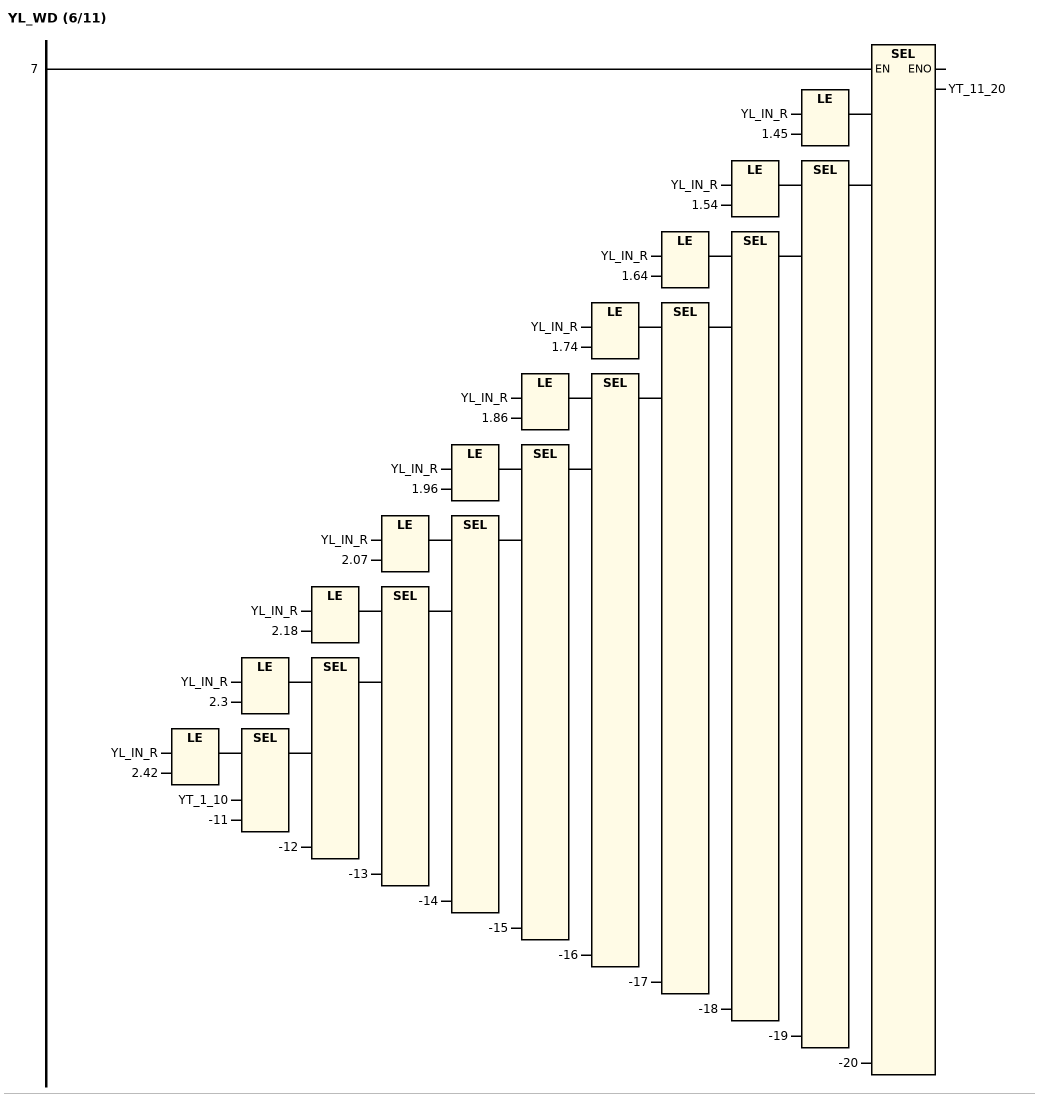
[picture p48: YL_WD (LD)]
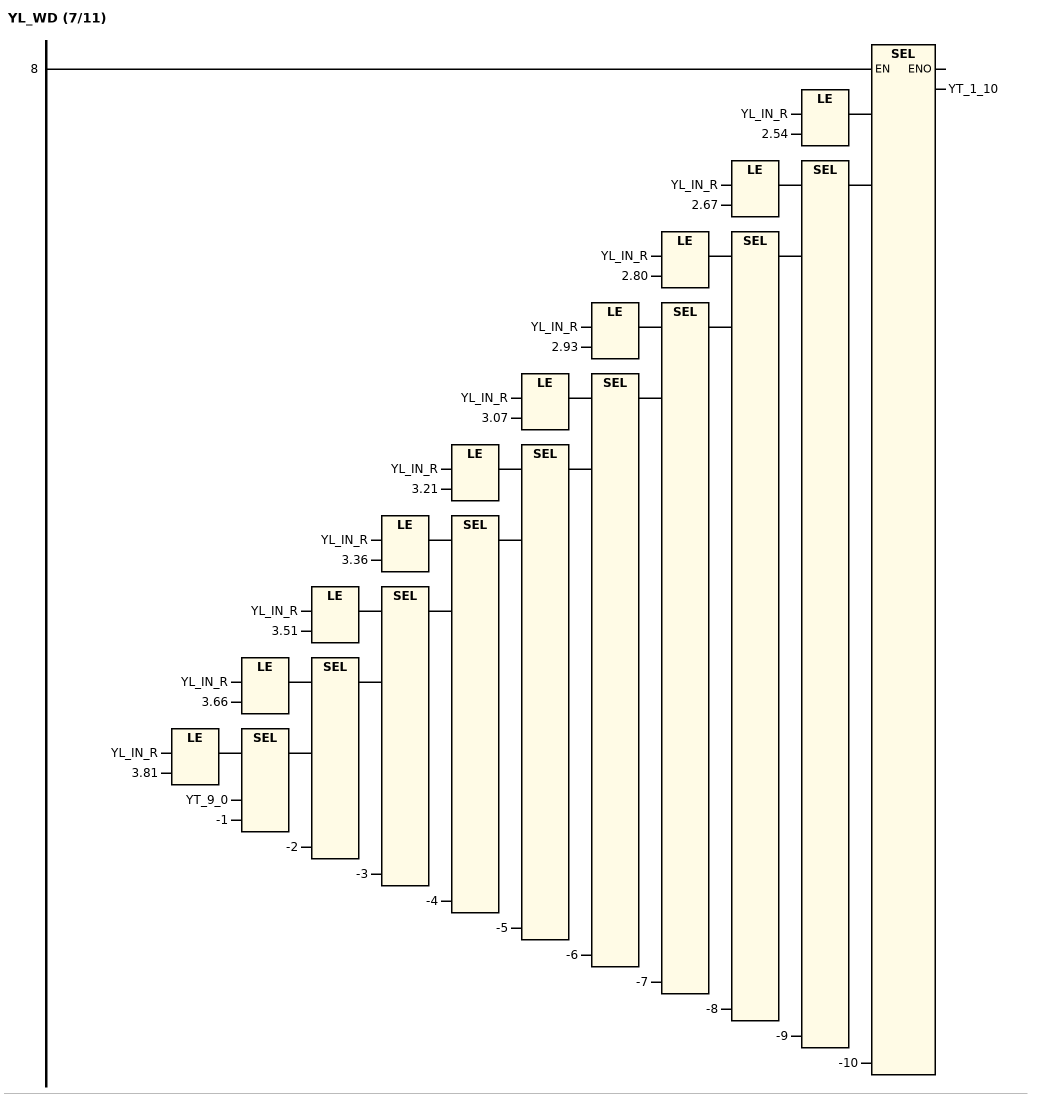
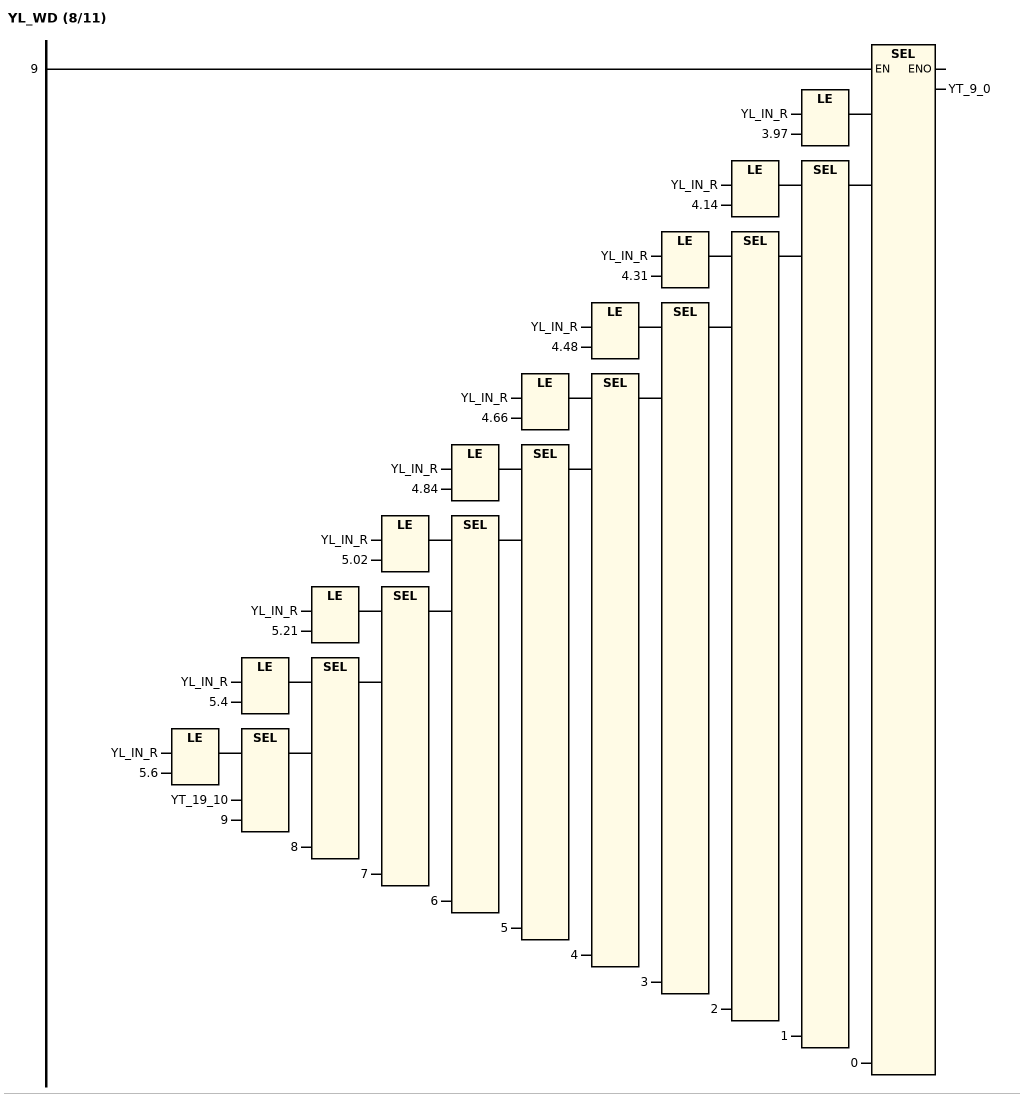
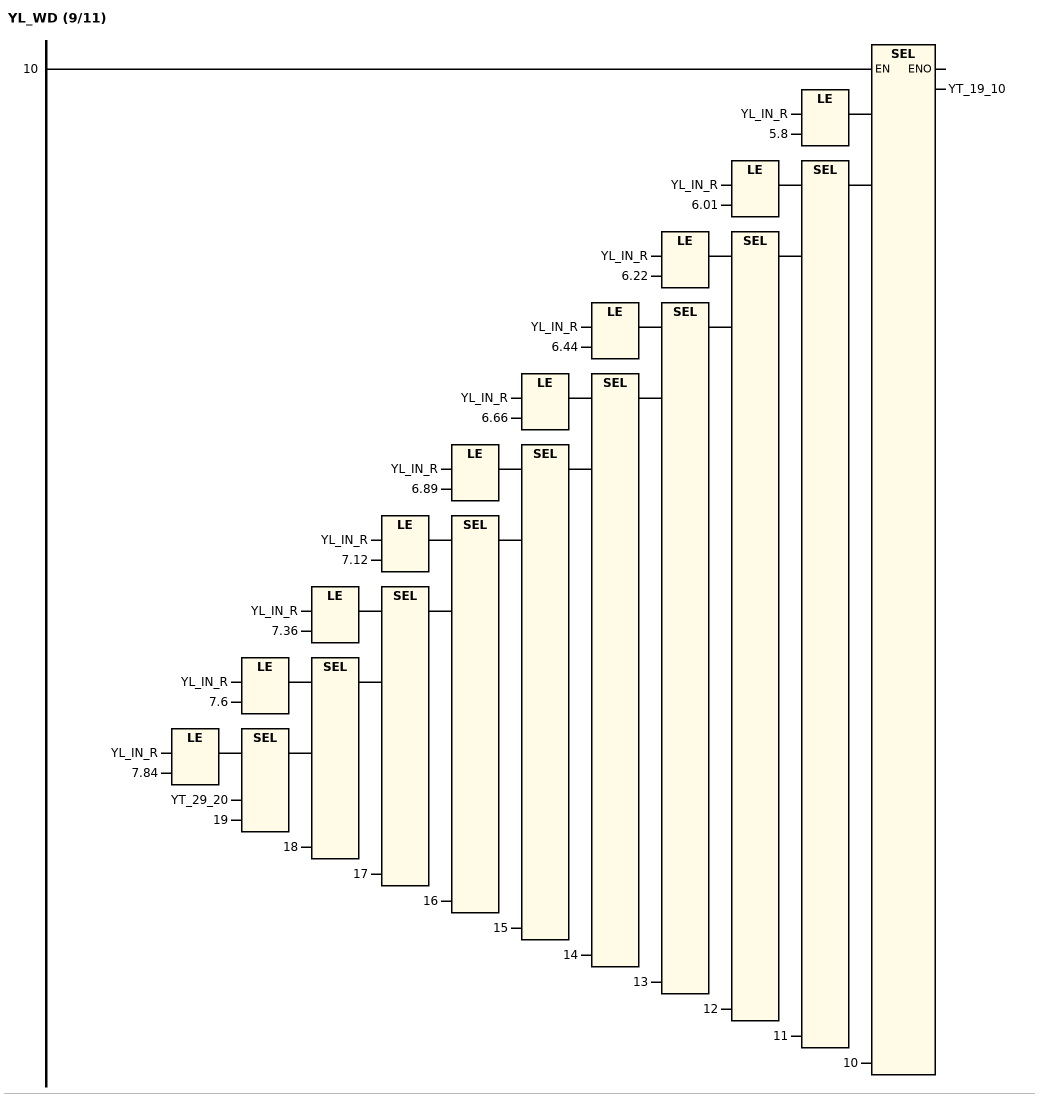
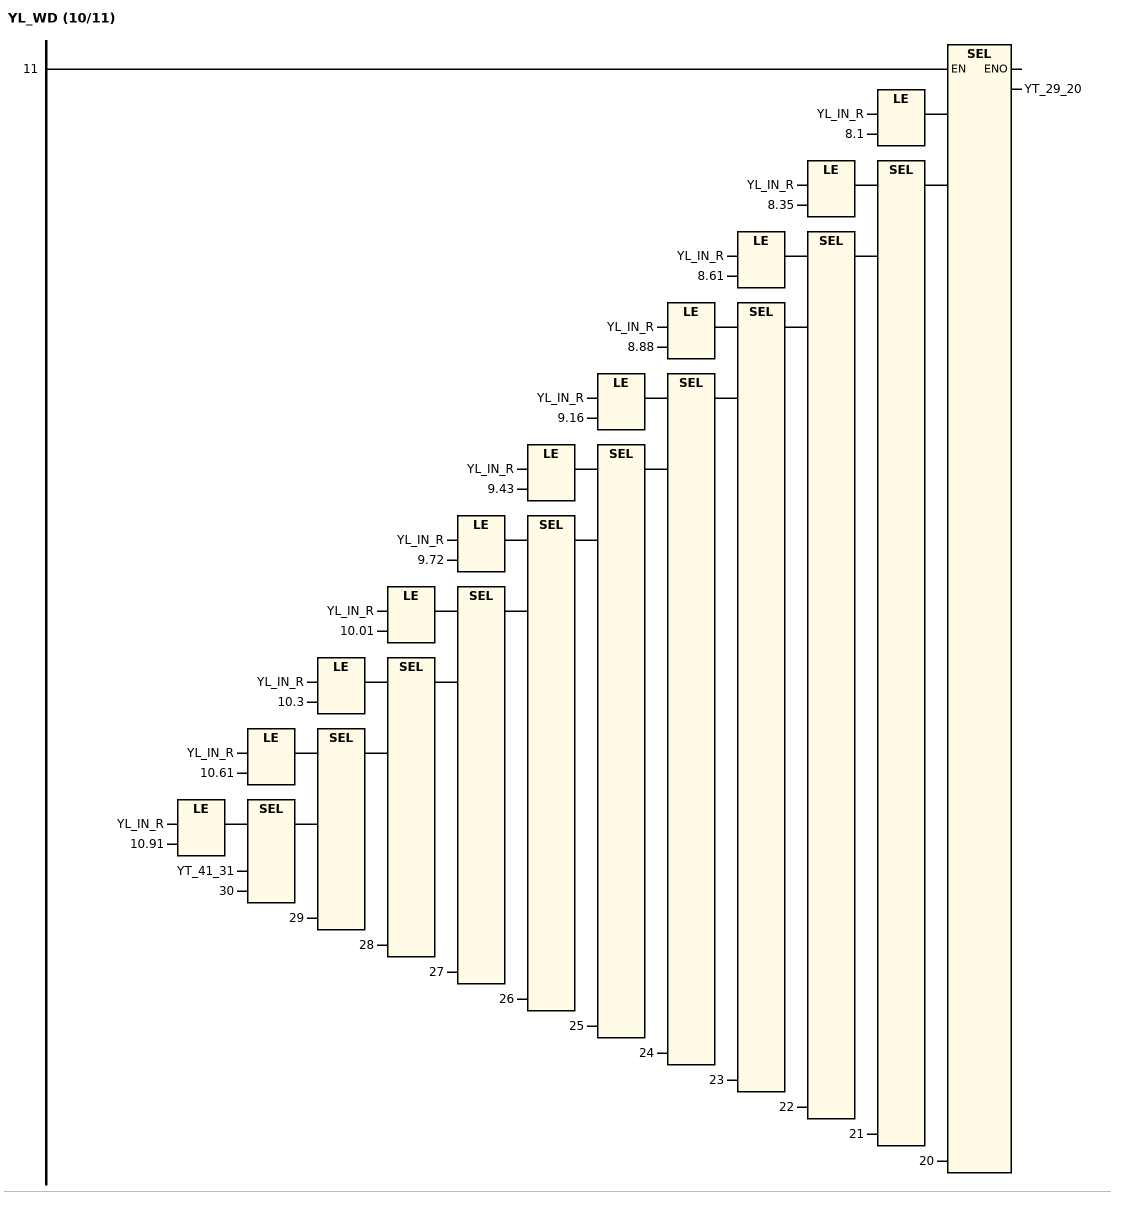
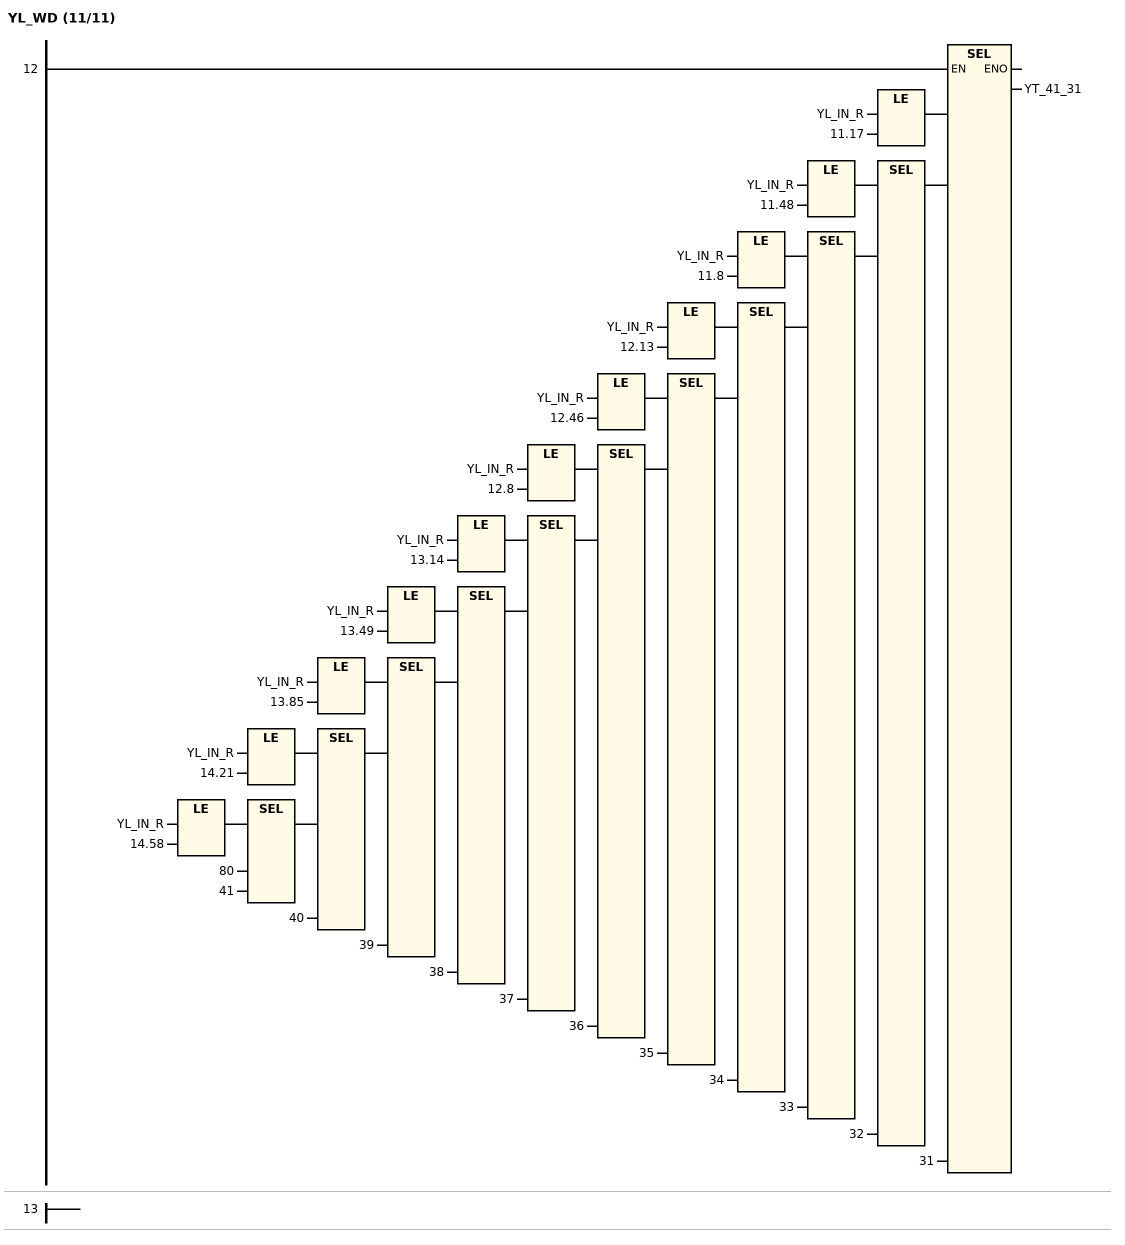
_LD_ (* Ladder Diagram *)
NETWORK 1
	*
		EN --- DIV(INT_TO_REAL(YL_IN), 100) => YL_IN_R
NETWORK 2
	*
		EN --- MUL(YL_T_KA, 10) => YL_T
NETWORK 3
	*
		EN --- SEL(LE(YL_IN_R, -0.62), SEL(LE(YL_IN_R, -0.60), SEL(LE(YL_IN_R, -0.58), SEL(LE(YL_IN_R, -0.55), SEL(LE(YL_IN_R, -0.53), SEL(LE(YL_IN_R, -0.50), SEL(LE(YL_IN_R, -0.46), SEL(LE(YL_IN_R, -0.44), SEL(LE(YL_IN_R, -0.41), SEL(LE(YL_IN_R, -0.38), YT_51_60, -51), -52), -53), -54), -55), -56), -57), -58), -59), -60) => YL_T_KA
NETWORK 4
	*
		EN --- SEL(LE(YL_IN_R, -0.35), SEL(LE(YL_IN_R, -0.32), SEL(LE(YL_IN_R, -0.28), SEL(LE(YL_IN_R, -0.24), SEL(LE(YL_IN_R, -0.21), SEL(LE(YL_IN_R, -0.17), SEL(LE(YL_IN_R, -0.12), SEL(LE(YL_IN_R, -0.08), SEL(LE(YL_IN_R, -0.04), SEL(LE(YL_IN_R, 0.00), YT_41_50, -41), -42), -43), -44), -45), -46), -47), -48), -49), -50) => YT_51_60
NETWORK 5
	*
		EN --- SEL(LE(YL_IN_R, 0.05), SEL(LE(YL_IN_R, 0.1), SEL(LE(YL_IN_R, 0.15), SEL(LE(YL_IN_R, 0.2), SEL(LE(YL_IN_R, 0.26), SEL(LE(YL_IN_R, 0.32), SEL(LE(YL_IN_R, 0.37), SEL(LE(YL_IN_R, 0.44), SEL(LE(YL_IN_R, 0.5), SEL(LE(YL_IN_R, 0.57), YT_31_40, -31), -32), -33), -34), -35), -36), -37), -38), -39), -40) => YT_41_50
NETWORK 6
	*
		EN --- SEL(LE(YL_IN_R, 0.63), SEL(LE(YL_IN_R, 0.70), SEL(LE(YL_IN_R, 0.78), SEL(LE(YL_IN_R, 0.85), SEL(LE(YL_IN_R, 0.93), SEL(LE(YL_IN_R, 1.01), SEL(LE(YL_IN_R, 1.09), SEL(LE(YL_IN_R, 1.18), SEL(LE(YL_IN_R, 1.26), SEL(LE(YL_IN_R, 1.36), YT_11_20, -21), -22), -23), -24), -25), -26), -27), -28), -29), -30) => YT_31_40
NETWORK 7
	*
		EN --- SEL(LE(YL_IN_R, 1.45), SEL(LE(YL_IN_R, 1.54), SEL(LE(YL_IN_R, 1.64), SEL(LE(YL_IN_R, 1.74), SEL(LE(YL_IN_R, 1.86), SEL(LE(YL_IN_R, 1.96), SEL(LE(YL_IN_R, 2.07), SEL(LE(YL_IN_R, 2.18), SEL(LE(YL_IN_R, 2.3), SEL(LE(YL_IN_R, 2.42), YT_1_10, -11), -12), -13), -14), -15), -16), -17), -18), -19), -20) => YT_11_20
NETWORK 8
	*
		EN --- SEL(LE(YL_IN_R, 2.54), SEL(LE(YL_IN_R, 2.67), SEL(LE(YL_IN_R, 2.80), SEL(LE(YL_IN_R, 2.93), SEL(LE(YL_IN_R, 3.07), SEL(LE(YL_IN_R, 3.21), SEL(LE(YL_IN_R, 3.36), SEL(LE(YL_IN_R, 3.51), SEL(LE(YL_IN_R, 3.66), SEL(LE(YL_IN_R, 3.81), YT_9_0, -1), -2), -3), -4), -5), -6), -7), -8), -9), -10) => YT_1_10
NETWORK 9
	*
		EN --- SEL(LE(YL_IN_R, 3.97), SEL(LE(YL_IN_R, 4.14), SEL(LE(YL_IN_R, 4.31), SEL(LE(YL_IN_R, 4.48), SEL(LE(YL_IN_R, 4.66), SEL(LE(YL_IN_R, 4.84), SEL(LE(YL_IN_R, 5.02), SEL(LE(YL_IN_R, 5.21), SEL(LE(YL_IN_R, 5.4), SEL(LE(YL_IN_R, 5.6), YT_19_10, 9), 8), 7), 6), 5), 4), 3), 2), 1), 0) => YT_9_0
NETWORK 10
	*
		EN --- SEL(LE(YL_IN_R, 5.8), SEL(LE(YL_IN_R, 6.01), SEL(LE(YL_IN_R, 6.22), SEL(LE(YL_IN_R, 6.44), SEL(LE(YL_IN_R, 6.66), SEL(LE(YL_IN_R, 6.89), SEL(LE(YL_IN_R, 7.12), SEL(LE(YL_IN_R, 7.36), SEL(LE(YL_IN_R, 7.6), SEL(LE(YL_IN_R, 7.84), YT_29_20, 19), 18), 17), 16), 15), 14), 13), 12), 11), 10) => YT_19_10
NETWORK 11
	*
		EN --- SEL(LE(YL_IN_R, 8.1), SEL(LE(YL_IN_R, 8.35), SEL(LE(YL_IN_R, 8.61), SEL(LE(YL_IN_R, 8.88), SEL(LE(YL_IN_R, 9.16), SEL(LE(YL_IN_R, 9.43), SEL(LE(YL_IN_R, 9.72), SEL(LE(YL_IN_R, 10.01), SEL(LE(YL_IN_R, 10.3), SEL(LE(YL_IN_R, 10.61), SEL(LE(YL_IN_R, 10.91), YT_41_31, 30), 29), 28), 27), 26), 25), 24), 23), 22), 21), 20) => YT_29_20
NETWORK 12
	*
		EN --- SEL(LE(YL_IN_R, 11.17), SEL(LE(YL_IN_R, 11.48), SEL(LE(YL_IN_R, 11.8), SEL(LE(YL_IN_R, 12.13), SEL(LE(YL_IN_R, 12.46), SEL(LE(YL_IN_R, 12.8), SEL(LE(YL_IN_R, 13.14), SEL(LE(YL_IN_R, 13.49), SEL(LE(YL_IN_R, 13.85), SEL(LE(YL_IN_R, 14.21), SEL(LE(YL_IN_R, 14.58), 80, 41), 40), 39), 38), 37), 36), 35), 34), 33), 32), 31) => YT_41_31
NETWORK 13
	*
_END_LD_
(* the same logic as Structured Text *)
(* Network 1 *)
YL_IN_R := INT_TO_REAL(YL_IN) / 100;
(* Network 2 *)
YL_T := YL_T_KA * 10;
(* Network 3 *)
YL_T_KA := SEL(YL_IN_R <= (-0.62), SEL(YL_IN_R <= (-0.60), SEL(YL_IN_R <= (-0.58), SEL(YL_IN_R <= (-0.55), SEL(YL_IN_R <= (-0.53), SEL(YL_IN_R <= (-0.50), SEL(YL_IN_R <= (-0.46), SEL(YL_IN_R <= (-0.44), SEL(YL_IN_R <= (-0.41), SEL(YL_IN_R <= (-0.38), YT_51_60, -51), -52), -53), -54), -55), -56), -57), -58), -59), -60);
(* Network 4 *)
YT_51_60 := SEL(YL_IN_R <= (-0.35), SEL(YL_IN_R <= (-0.32), SEL(YL_IN_R <= (-0.28), SEL(YL_IN_R <= (-0.24), SEL(YL_IN_R <= (-0.21), SEL(YL_IN_R <= (-0.17), SEL(YL_IN_R <= (-0.12), SEL(YL_IN_R <= (-0.08), SEL(YL_IN_R <= (-0.04), SEL(YL_IN_R <= 0.00, YT_41_50, -41), -42), -43), -44), -45), -46), -47), -48), -49), -50);
(* Network 5 *)
YT_41_50 := SEL(YL_IN_R <= 0.05, SEL(YL_IN_R <= 0.1, SEL(YL_IN_R <= 0.15, SEL(YL_IN_R <= 0.2, SEL(YL_IN_R <= 0.26, SEL(YL_IN_R <= 0.32, SEL(YL_IN_R <= 0.37, SEL(YL_IN_R <= 0.44, SEL(YL_IN_R <= 0.5, SEL(YL_IN_R <= 0.57, YT_31_40, -31), -32), -33), -34), -35), -36), -37), -38), -39), -40);
(* Network 6 *)
YT_31_40 := SEL(YL_IN_R <= 0.63, SEL(YL_IN_R <= 0.70, SEL(YL_IN_R <= 0.78, SEL(YL_IN_R <= 0.85, SEL(YL_IN_R <= 0.93, SEL(YL_IN_R <= 1.01, SEL(YL_IN_R <= 1.09, SEL(YL_IN_R <= 1.18, SEL(YL_IN_R <= 1.26, SEL(YL_IN_R <= 1.36, YT_11_20, -21), -22), -23), -24), -25), -26), -27), -28), -29), -30);
(* Network 7 *)
YT_11_20 := SEL(YL_IN_R <= 1.45, SEL(YL_IN_R <= 1.54, SEL(YL_IN_R <= 1.64, SEL(YL_IN_R <= 1.74, SEL(YL_IN_R <= 1.86, SEL(YL_IN_R <= 1.96, SEL(YL_IN_R <= 2.07, SEL(YL_IN_R <= 2.18, SEL(YL_IN_R <= 2.3, SEL(YL_IN_R <= 2.42, YT_1_10, -11), -12), -13), -14), -15), -16), -17), -18), -19), -20);
(* Network 8 *)
YT_1_10 := SEL(YL_IN_R <= 2.54, SEL(YL_IN_R <= 2.67, SEL(YL_IN_R <= 2.80, SEL(YL_IN_R <= 2.93, SEL(YL_IN_R <= 3.07, SEL(YL_IN_R <= 3.21, SEL(YL_IN_R <= 3.36, SEL(YL_IN_R <= 3.51, SEL(YL_IN_R <= 3.66, SEL(YL_IN_R <= 3.81, YT_9_0, -1), -2), -3), -4), -5), -6), -7), -8), -9), -10);
(* Network 9 *)
YT_9_0 := SEL(YL_IN_R <= 3.97, SEL(YL_IN_R <= 4.14, SEL(YL_IN_R <= 4.31, SEL(YL_IN_R <= 4.48, SEL(YL_IN_R <= 4.66, SEL(YL_IN_R <= 4.84, SEL(YL_IN_R <= 5.02, SEL(YL_IN_R <= 5.21, SEL(YL_IN_R <= 5.4, SEL(YL_IN_R <= 5.6, YT_19_10, 9), 8), 7), 6), 5), 4), 3), 2), 1), 0);
(* Network 10 *)
YT_19_10 := SEL(YL_IN_R <= 5.8, SEL(YL_IN_R <= 6.01, SEL(YL_IN_R <= 6.22, SEL(YL_IN_R <= 6.44, SEL(YL_IN_R <= 6.66, SEL(YL_IN_R <= 6.89, SEL(YL_IN_R <= 7.12, SEL(YL_IN_R <= 7.36, SEL(YL_IN_R <= 7.6, SEL(YL_IN_R <= 7.84, YT_29_20, 19), 18), 17), 16), 15), 14), 13), 12), 11), 10);
(* Network 11 *)
YT_29_20 := SEL(YL_IN_R <= 8.1, SEL(YL_IN_R <= 8.35, SEL(YL_IN_R <= 8.61, SEL(YL_IN_R <= 8.88, SEL(YL_IN_R <= 9.16, SEL(YL_IN_R <= 9.43, SEL(YL_IN_R <= 9.72, SEL(YL_IN_R <= 10.01, SEL(YL_IN_R <= 10.3, SEL(YL_IN_R <= 10.61, SEL(YL_IN_R <= 10.91, YT_41_31, 30), 29), 28), 27), 26), 25), 24), 23), 22), 21), 20);
(* Network 12 *)
YT_41_31 := SEL(YL_IN_R <= 11.17, SEL(YL_IN_R <= 11.48, SEL(YL_IN_R <= 11.8, SEL(YL_IN_R <= 12.13, SEL(YL_IN_R <= 12.46, SEL(YL_IN_R <= 12.8, SEL(YL_IN_R <= 13.14, SEL(YL_IN_R <= 13.49, SEL(YL_IN_R <= 13.85, SEL(YL_IN_R <= 14.21, SEL(YL_IN_R <= 14.58, 80, 41), 40), 39), 38), 37), 36), 35), 34), 33), 32), 31);
(* Network 13 *)
END_FUNCTION_BLOCK

(* POU BJ_MIN_COOL, LD *)
FUNCTION_BLOCK BJ_MIN_COOL
VAR_INPUT
	XH_SHU: WORD;
	ONE_H_IN: DWORD;
	TWO_H_IN: DWORD;
	THREE_H_IN: DWORD;
	FOUER_H_IN: DWORD;
	FIVE_H_IN: DWORD;
	SIX_H_IN: DWORD;
	CHD_ONE_IN: BOOL;
	CHD_TWO_IN: BOOL;
	CHD_THREE_IN: BOOL;
	CHD_FOUER_IN: BOOL;
	CHD_FIVE_IN: BOOL;
	CHD_SIX_IN: BOOL;
	FUWEI_KZH: BOOL;
END_VAR
VAR_OUTPUT
	ONE_CIXU: BYTE;
	TWO_CIXU: BYTE;
	THREE_CIXU: BYTE;
	FOUER_CIXU: BYTE;
	FIVE_CIXU: BYTE;
	SIX_CIXU: BYTE;
END_VAR
VAR
	ONE_H_ZC_1: DWORD;
	TWO_H_ZC_1: DWORD;
	THREE_H_ZC_1: DWORD;
	FOUER_H_ZC_1: DWORD;
	FIVE_H_ZC_1: DWORD;
	ONE_CX_ZC: BYTE;
	TWO_CX_ZC: BYTE;
	THREE_CX_ZC: BYTE;
	FOUER_CX_ZC: BYTE;
	FIVE_CX_ZC: BYTE;
	ONE_H_ZC_2: DWORD;
	TWO_H_ZC_2: DWORD;
	THREE_H_ZC_2: DWORD;
	FOUER_H_ZC_2: DWORD;
	FIVE_H_ZC_2: DWORD;
	ONE_FUWEI: BOOL;
	TWO_FUWEI: BOOL;
	FIVE_FUWEI: BOOL;
	FOUER_FUWEI: BOOL;
	THREE_FUWEI: BOOL;
	R1_IN: R_TRIG;
	BJ_COOL: BJ_CIXU_COOL;
	XH_SHU_1: BOOL;
	SIX_FUWEI: BOOL;
	SIX_H_ZC_1: DWORD;
	SIX_H_ZC_2: DWORD;
	SIX_CX_ZC: BYTE;
END_VAR
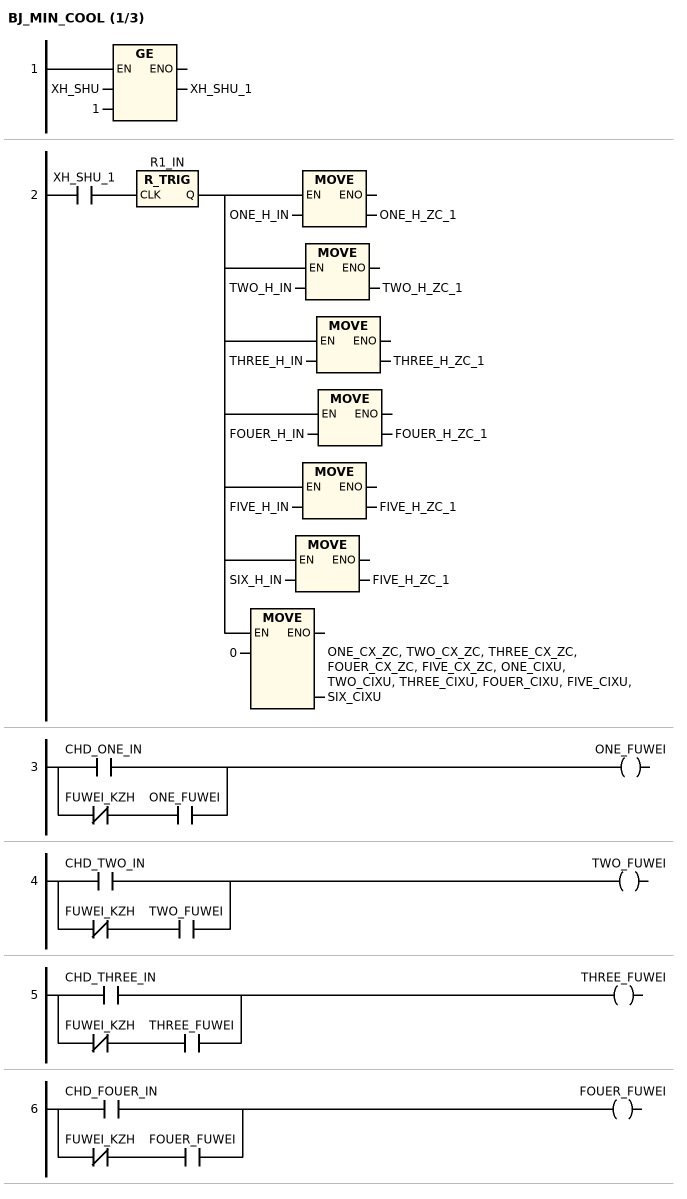
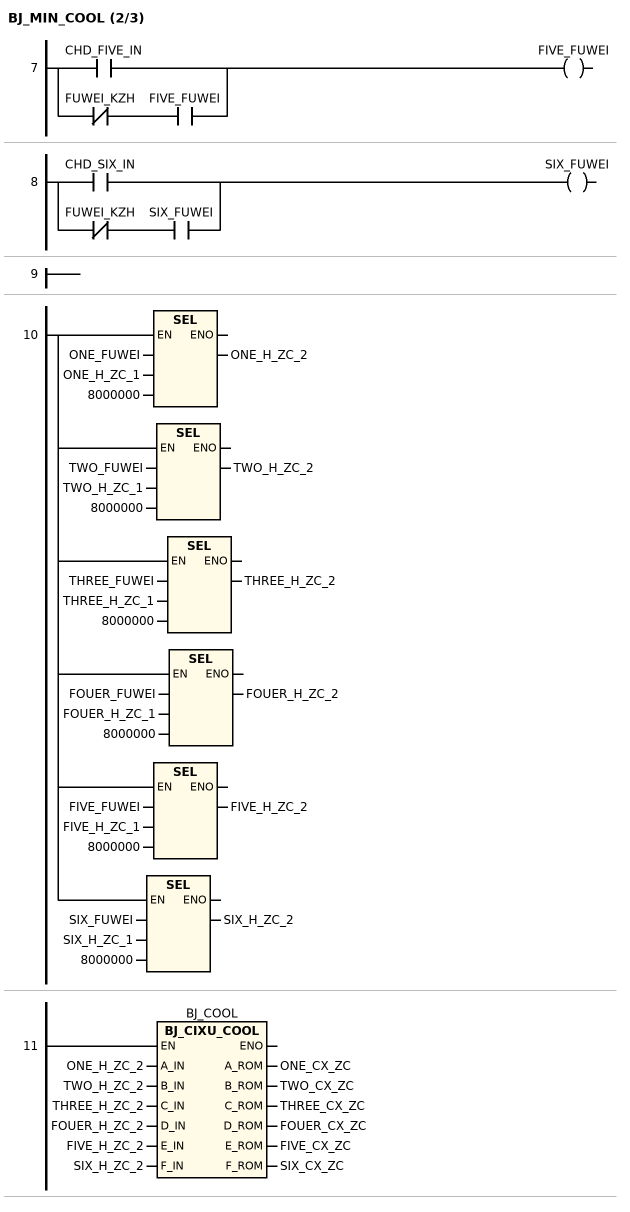
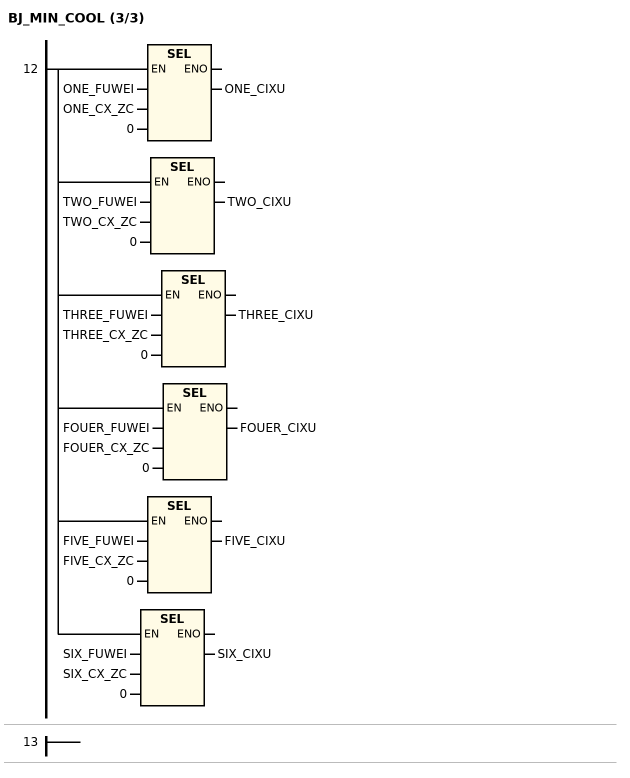
_LD_ (* Ladder Diagram *)
NETWORK 1
	*
		EN --- GE(XH_SHU, 1) => XH_SHU_1
NETWORK 2
	[XH_SHU_1] - R1_IN:R_TRIG(CLK: *)
		EN --- MOVE(ONE_H_IN) => ONE_H_ZC_1
		EN --- MOVE(TWO_H_IN) => TWO_H_ZC_1
		EN --- MOVE(THREE_H_IN) => THREE_H_ZC_1
		EN --- MOVE(FOUER_H_IN) => FOUER_H_ZC_1
		EN --- MOVE(FIVE_H_IN) => FIVE_H_ZC_1
		EN --- MOVE(SIX_H_IN) => FIVE_H_ZC_1
		EN --- MOVE(0) => ONE_CX_ZC, TWO_CX_ZC, THREE_CX_ZC, FOUER_CX_ZC, FIVE_CX_ZC, ONE_CIXU, TWO_CIXU, THREE_CIXU, FOUER_CIXU, FIVE_CIXU, SIX_CIXU
NETWORK 3
	{ [CHD_ONE_IN] | [/FUWEI_KZH] - [ONE_FUWEI] } --- (ONE_FUWEI)
NETWORK 4
	{ [CHD_TWO_IN] | [/FUWEI_KZH] - [TWO_FUWEI] } --- (TWO_FUWEI)
NETWORK 5
	{ [CHD_THREE_IN] | [/FUWEI_KZH] - [THREE_FUWEI] } --- (THREE_FUWEI)
NETWORK 6
	{ [CHD_FOUER_IN] | [/FUWEI_KZH] - [FOUER_FUWEI] } --- (FOUER_FUWEI)
NETWORK 7
	{ [CHD_FIVE_IN] | [/FUWEI_KZH] - [FIVE_FUWEI] } --- (FIVE_FUWEI)
NETWORK 8
	{ [CHD_SIX_IN] | [/FUWEI_KZH] - [SIX_FUWEI] } --- (SIX_FUWEI)
NETWORK 9
	*
NETWORK 10
	*
		EN --- SEL(ONE_FUWEI, ONE_H_ZC_1, 8000000) => ONE_H_ZC_2
		EN --- SEL(TWO_FUWEI, TWO_H_ZC_1, 8000000) => TWO_H_ZC_2
		EN --- SEL(THREE_FUWEI, THREE_H_ZC_1, 8000000) => THREE_H_ZC_2
		EN --- SEL(FOUER_FUWEI, FOUER_H_ZC_1, 8000000) => FOUER_H_ZC_2
		EN --- SEL(FIVE_FUWEI, FIVE_H_ZC_1, 8000000) => FIVE_H_ZC_2
		EN --- SEL(SIX_FUWEI, SIX_H_ZC_1, 8000000) => SIX_H_ZC_2
NETWORK 11
	*
		EN --- BJ_COOL:BJ_CIXU_COOL(A_IN: ONE_H_ZC_2, B_IN: TWO_H_ZC_2, C_IN: THREE_H_ZC_2, D_IN: FOUER_H_ZC_2, E_IN: FIVE_H_ZC_2, F_IN: SIX_H_ZC_2, B_ROM => TWO_CX_ZC, C_ROM => THREE_CX_ZC, D_ROM => FOUER_CX_ZC, E_ROM => FIVE_CX_ZC, F_ROM => SIX_CX_ZC) => ONE_CX_ZC
NETWORK 12
	*
		EN --- SEL(ONE_FUWEI, ONE_CX_ZC, 0) => ONE_CIXU
		EN --- SEL(TWO_FUWEI, TWO_CX_ZC, 0) => TWO_CIXU
		EN --- SEL(THREE_FUWEI, THREE_CX_ZC, 0) => THREE_CIXU
		EN --- SEL(FOUER_FUWEI, FOUER_CX_ZC, 0) => FOUER_CIXU
		EN --- SEL(FIVE_FUWEI, FIVE_CX_ZC, 0) => FIVE_CIXU
		EN --- SEL(SIX_FUWEI, SIX_CX_ZC, 0) => SIX_CIXU
NETWORK 13
	*
_END_LD_
(* the same logic as Structured Text *)
(* Network 1 *)
XH_SHU_1 := XH_SHU >= 1;
(* Network 2: see the listing above *)
(* Network 3 *)
ONE_FUWEI := CHD_ONE_IN OR NOT FUWEI_KZH AND ONE_FUWEI;
(* Network 4 *)
TWO_FUWEI := CHD_TWO_IN OR NOT FUWEI_KZH AND TWO_FUWEI;
(* Network 5 *)
THREE_FUWEI := CHD_THREE_IN OR NOT FUWEI_KZH AND THREE_FUWEI;
(* Network 6 *)
FOUER_FUWEI := CHD_FOUER_IN OR NOT FUWEI_KZH AND FOUER_FUWEI;
(* Network 7 *)
FIVE_FUWEI := CHD_FIVE_IN OR NOT FUWEI_KZH AND FIVE_FUWEI;
(* Network 8 *)
SIX_FUWEI := CHD_SIX_IN OR NOT FUWEI_KZH AND SIX_FUWEI;
(* Network 9: see the listing above *)
(* Network 10 *)
ONE_H_ZC_2 := SEL(ONE_FUWEI, ONE_H_ZC_1, 8000000);
TWO_H_ZC_2 := SEL(TWO_FUWEI, TWO_H_ZC_1, 8000000);
THREE_H_ZC_2 := SEL(THREE_FUWEI, THREE_H_ZC_1, 8000000);
FOUER_H_ZC_2 := SEL(FOUER_FUWEI, FOUER_H_ZC_1, 8000000);
FIVE_H_ZC_2 := SEL(FIVE_FUWEI, FIVE_H_ZC_1, 8000000);
SIX_H_ZC_2 := SEL(SIX_FUWEI, SIX_H_ZC_1, 8000000);
(* Network 11 *)
BJ_COOL(A_IN := ONE_H_ZC_2, B_IN := TWO_H_ZC_2, C_IN := THREE_H_ZC_2, D_IN := FOUER_H_ZC_2, E_IN := FIVE_H_ZC_2, F_IN := SIX_H_ZC_2);
TWO_CX_ZC := BJ_COOL.B_ROM;
THREE_CX_ZC := BJ_COOL.C_ROM;
FOUER_CX_ZC := BJ_COOL.D_ROM;
FIVE_CX_ZC := BJ_COOL.E_ROM;
SIX_CX_ZC := BJ_COOL.F_ROM;
ONE_CX_ZC := BJ_COOL.A_ROM;
(* Network 12 *)
ONE_CIXU := SEL(ONE_FUWEI, ONE_CX_ZC, 0);
TWO_CIXU := SEL(TWO_FUWEI, TWO_CX_ZC, 0);
THREE_CIXU := SEL(THREE_FUWEI, THREE_CX_ZC, 0);
FOUER_CIXU := SEL(FOUER_FUWEI, FOUER_CX_ZC, 0);
FIVE_CIXU := SEL(FIVE_FUWEI, FIVE_CX_ZC, 0);
SIX_CIXU := SEL(SIX_FUWEI, SIX_CX_ZC, 0);
(* Network 13: see the listing above *)
END_FUNCTION_BLOCK

(* POU BJ_CIXU_COOL, LD *)
FUNCTION_BLOCK BJ_CIXU_COOL
VAR_INPUT
	A_IN:DWORD;
	B_IN: DWORD;
	C_IN: DWORD;
	D_IN: DWORD;
	E_IN: DWORD;
	F_IN: DWORD;
END_VAR
VAR_OUTPUT
	A_ROM: BYTE;
	B_ROM: BYTE;
	C_ROM: BYTE;
	D_ROM: BYTE;
	E_ROM: BYTE;
	F_ROM: BYTE;
END_VAR
VAR
	A_B_OUT: BOOL;
	A_C_OUT: BOOL;
	A_D_OUT: BOOL;
	A_E_OUT: BOOL;
	B_A_OUT: BOOL;
	B_C_OUT: BOOL;
	B_D_OUT: BOOL;
	B_E_OUT: BOOL;
	C_A_OUT: BOOL;
	C_B_OUT: BOOL;
	C_D_OUT: BOOL;
	C_E_OUT: BOOL;
	D_E_OUT: BOOL;
	D_C_OUT: BOOL;
	D_B_OUT: BOOL;
	D_A_OUT: BOOL;
	E_A_OUT: BOOL;
	E_B_OUT: BOOL;
	E_C_OUT: BOOL;
	E_D_OUT: BOOL;

	A_F_OUT: BOOL;
	B_F_OUT: BOOL;
	C_F_OUT: BOOL;
	D_F_OUT: BOOL;
	E_F_OUT: BOOL;
	F_A_OUT: BOOL;
	F_B_OUT: BOOL;
	F_C_OUT: BOOL;
	F_D_OUT: BOOL;

	F_E_OUT: BOOL;
END_VAR
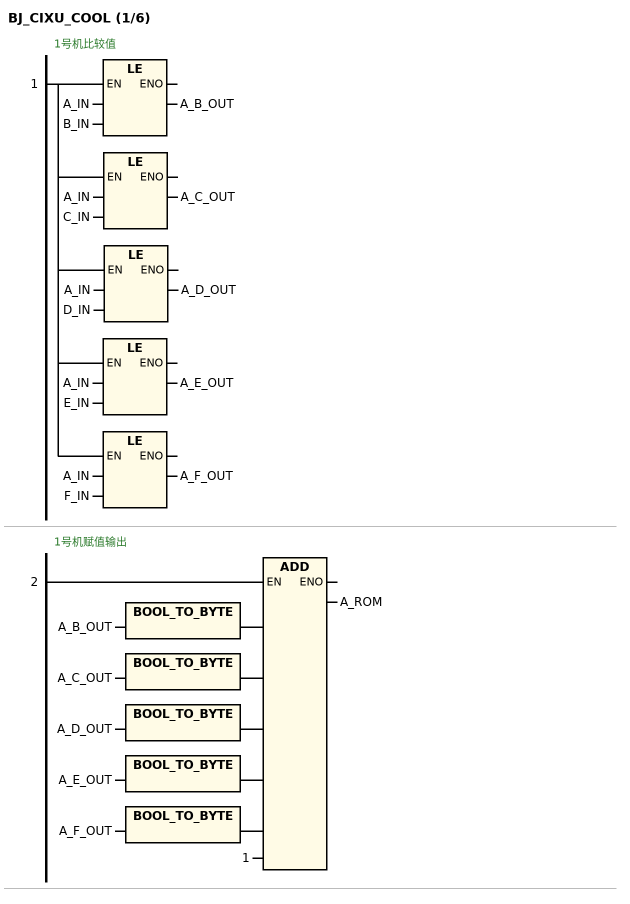
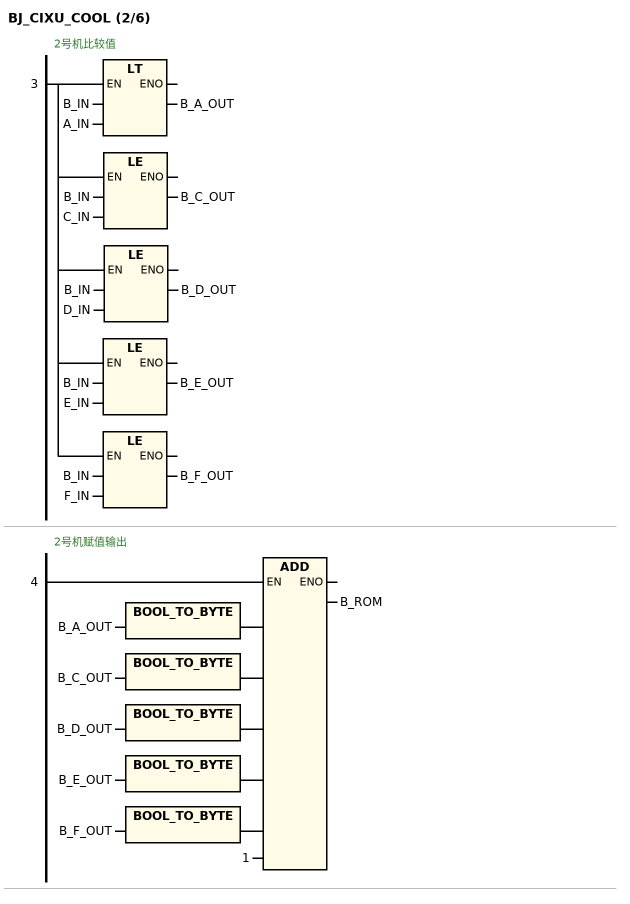
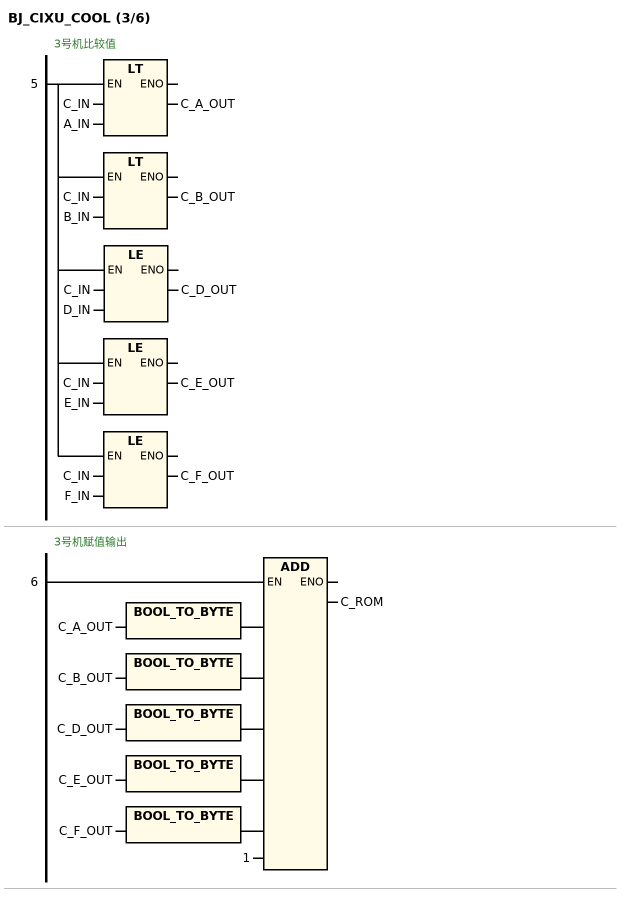
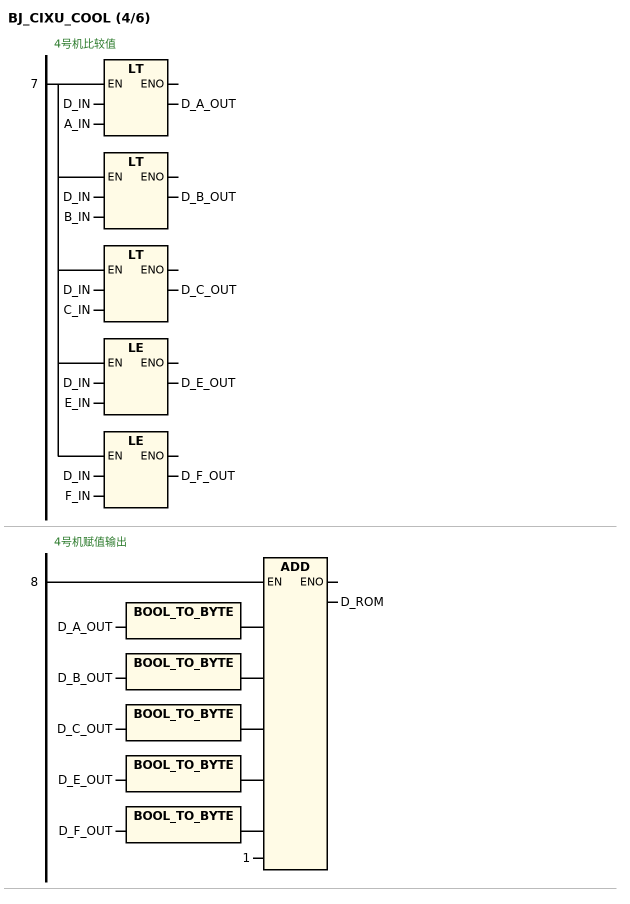
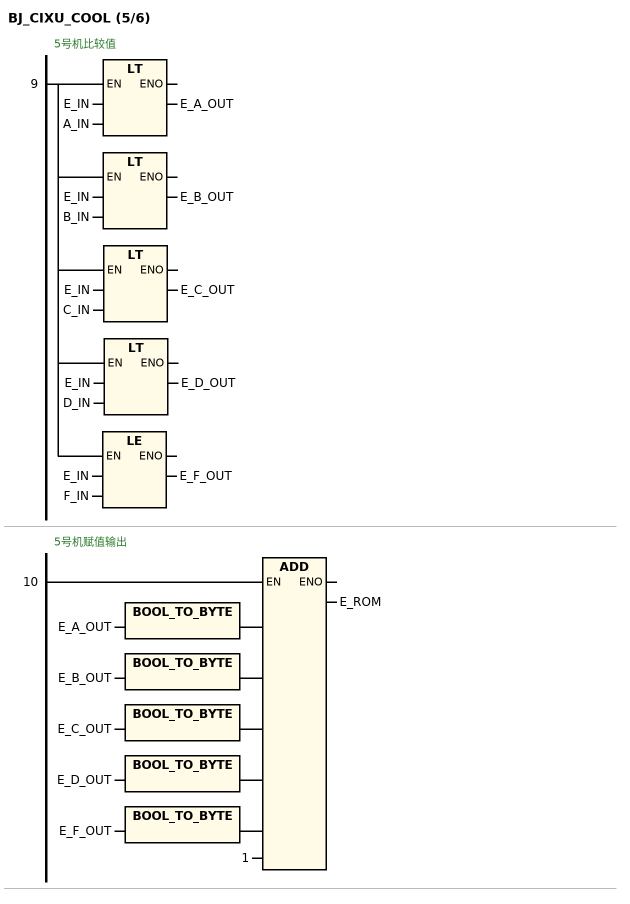
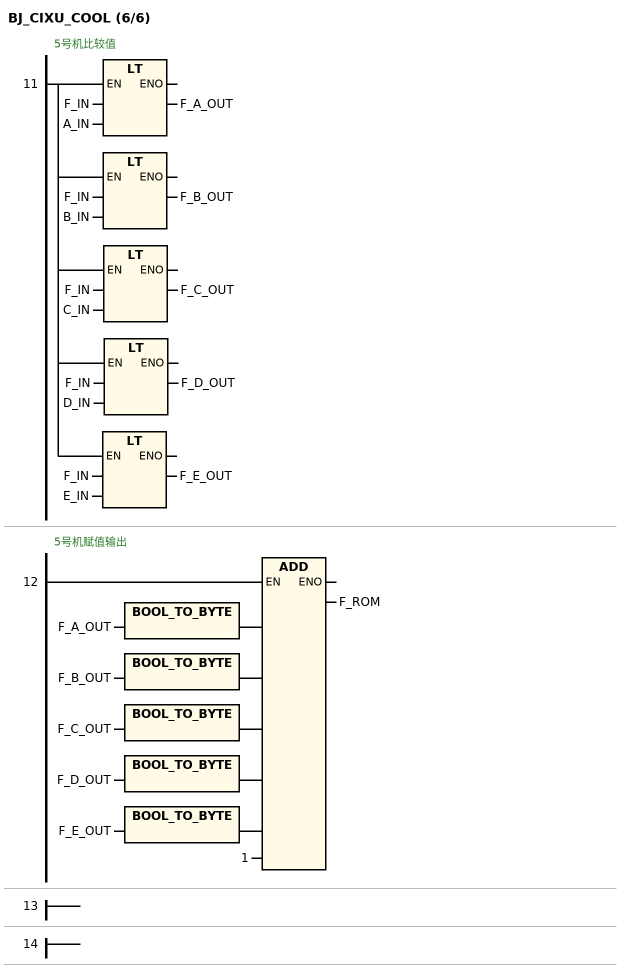
_LD_ (* Ladder Diagram *)
NETWORK 1 (* 1号机比较值 *)
	*
		EN --- LE(A_IN, B_IN) => A_B_OUT
		EN --- LE(A_IN, C_IN) => A_C_OUT
		EN --- LE(A_IN, D_IN) => A_D_OUT
		EN --- LE(A_IN, E_IN) => A_E_OUT
		EN --- LE(A_IN, F_IN) => A_F_OUT
NETWORK 2 (* 1号机赋值输出 *)
	*
		EN --- ADD(BOOL_TO_BYTE(A_B_OUT), BOOL_TO_BYTE(A_C_OUT), BOOL_TO_BYTE(A_D_OUT), BOOL_TO_BYTE(A_E_OUT), BOOL_TO_BYTE(A_F_OUT), 1) => A_ROM
NETWORK 3 (* 2号机比较值 *)
	*
		EN --- LT(B_IN, A_IN) => B_A_OUT
		EN --- LE(B_IN, C_IN) => B_C_OUT
		EN --- LE(B_IN, D_IN) => B_D_OUT
		EN --- LE(B_IN, E_IN) => B_E_OUT
		EN --- LE(B_IN, F_IN) => B_F_OUT
NETWORK 4 (* 2号机赋值输出 *)
	*
		EN --- ADD(BOOL_TO_BYTE(B_A_OUT), BOOL_TO_BYTE(B_C_OUT), BOOL_TO_BYTE(B_D_OUT), BOOL_TO_BYTE(B_E_OUT), BOOL_TO_BYTE(B_F_OUT), 1) => B_ROM
NETWORK 5 (* 3号机比较值 *)
	*
		EN --- LT(C_IN, A_IN) => C_A_OUT
		EN --- LT(C_IN, B_IN) => C_B_OUT
		EN --- LE(C_IN, D_IN) => C_D_OUT
		EN --- LE(C_IN, E_IN) => C_E_OUT
		EN --- LE(C_IN, F_IN) => C_F_OUT
NETWORK 6 (* 3号机赋值输出 *)
	*
		EN --- ADD(BOOL_TO_BYTE(C_A_OUT), BOOL_TO_BYTE(C_B_OUT), BOOL_TO_BYTE(C_D_OUT), BOOL_TO_BYTE(C_E_OUT), BOOL_TO_BYTE(C_F_OUT), 1) => C_ROM
NETWORK 7 (* 4号机比较值 *)
	*
		EN --- LT(D_IN, A_IN) => D_A_OUT
		EN --- LT(D_IN, B_IN) => D_B_OUT
		EN --- LT(D_IN, C_IN) => D_C_OUT
		EN --- LE(D_IN, E_IN) => D_E_OUT
		EN --- LE(D_IN, F_IN) => D_F_OUT
NETWORK 8 (* 4号机赋值输出 *)
	*
		EN --- ADD(BOOL_TO_BYTE(D_A_OUT), BOOL_TO_BYTE(D_B_OUT), BOOL_TO_BYTE(D_C_OUT), BOOL_TO_BYTE(D_E_OUT), BOOL_TO_BYTE(D_F_OUT), 1) => D_ROM
NETWORK 9 (* 5号机比较值 *)
	*
		EN --- LT(E_IN, A_IN) => E_A_OUT
		EN --- LT(E_IN, B_IN) => E_B_OUT
		EN --- LT(E_IN, C_IN) => E_C_OUT
		EN --- LT(E_IN, D_IN) => E_D_OUT
		EN --- LE(E_IN, F_IN) => E_F_OUT
NETWORK 10 (* 5号机赋值输出 *)
	*
		EN --- ADD(BOOL_TO_BYTE(E_A_OUT), BOOL_TO_BYTE(E_B_OUT), BOOL_TO_BYTE(E_C_OUT), BOOL_TO_BYTE(E_D_OUT), BOOL_TO_BYTE(E_F_OUT), 1) => E_ROM
NETWORK 11 (* 5号机比较值 *)
	*
		EN --- LT(F_IN, A_IN) => F_A_OUT
		EN --- LT(F_IN, B_IN) => F_B_OUT
		EN --- LT(F_IN, C_IN) => F_C_OUT
		EN --- LT(F_IN, D_IN) => F_D_OUT
		EN --- LT(F_IN, E_IN) => F_E_OUT
NETWORK 12 (* 5号机赋值输出 *)
	*
		EN --- ADD(BOOL_TO_BYTE(F_A_OUT), BOOL_TO_BYTE(F_B_OUT), BOOL_TO_BYTE(F_C_OUT), BOOL_TO_BYTE(F_D_OUT), BOOL_TO_BYTE(F_E_OUT), 1) => F_ROM
NETWORK 13
	*
NETWORK 14
	*
_END_LD_
(* the same logic as Structured Text *)
(* Network 1: 1号机比较值 *)
A_B_OUT := A_IN <= B_IN;
A_C_OUT := A_IN <= C_IN;
A_D_OUT := A_IN <= D_IN;
A_E_OUT := A_IN <= E_IN;
A_F_OUT := A_IN <= F_IN;
(* Network 2: 1号机赋值输出 *)
A_ROM := BOOL_TO_BYTE(A_B_OUT) + BOOL_TO_BYTE(A_C_OUT) + BOOL_TO_BYTE(A_D_OUT) + BOOL_TO_BYTE(A_E_OUT) + BOOL_TO_BYTE(A_F_OUT) + 1;
(* Network 3: 2号机比较值 *)
B_A_OUT := B_IN < A_IN;
B_C_OUT := B_IN <= C_IN;
B_D_OUT := B_IN <= D_IN;
B_E_OUT := B_IN <= E_IN;
B_F_OUT := B_IN <= F_IN;
(* Network 4: 2号机赋值输出 *)
B_ROM := BOOL_TO_BYTE(B_A_OUT) + BOOL_TO_BYTE(B_C_OUT) + BOOL_TO_BYTE(B_D_OUT) + BOOL_TO_BYTE(B_E_OUT) + BOOL_TO_BYTE(B_F_OUT) + 1;
(* Network 5: 3号机比较值 *)
C_A_OUT := C_IN < A_IN;
C_B_OUT := C_IN < B_IN;
C_D_OUT := C_IN <= D_IN;
C_E_OUT := C_IN <= E_IN;
C_F_OUT := C_IN <= F_IN;
(* Network 6: 3号机赋值输出 *)
C_ROM := BOOL_TO_BYTE(C_A_OUT) + BOOL_TO_BYTE(C_B_OUT) + BOOL_TO_BYTE(C_D_OUT) + BOOL_TO_BYTE(C_E_OUT) + BOOL_TO_BYTE(C_F_OUT) + 1;
(* Network 7: 4号机比较值 *)
D_A_OUT := D_IN < A_IN;
D_B_OUT := D_IN < B_IN;
D_C_OUT := D_IN < C_IN;
D_E_OUT := D_IN <= E_IN;
D_F_OUT := D_IN <= F_IN;
(* Network 8: 4号机赋值输出 *)
D_ROM := BOOL_TO_BYTE(D_A_OUT) + BOOL_TO_BYTE(D_B_OUT) + BOOL_TO_BYTE(D_C_OUT) + BOOL_TO_BYTE(D_E_OUT) + BOOL_TO_BYTE(D_F_OUT) + 1;
(* Network 9: 5号机比较值 *)
E_A_OUT := E_IN < A_IN;
E_B_OUT := E_IN < B_IN;
E_C_OUT := E_IN < C_IN;
E_D_OUT := E_IN < D_IN;
E_F_OUT := E_IN <= F_IN;
(* Network 10: 5号机赋值输出 *)
E_ROM := BOOL_TO_BYTE(E_A_OUT) + BOOL_TO_BYTE(E_B_OUT) + BOOL_TO_BYTE(E_C_OUT) + BOOL_TO_BYTE(E_D_OUT) + BOOL_TO_BYTE(E_F_OUT) + 1;
(* Network 11: 5号机比较值 *)
F_A_OUT := F_IN < A_IN;
F_B_OUT := F_IN < B_IN;
F_C_OUT := F_IN < C_IN;
F_D_OUT := F_IN < D_IN;
F_E_OUT := F_IN < E_IN;
(* Network 12: 5号机赋值输出 *)
F_ROM := BOOL_TO_BYTE(F_A_OUT) + BOOL_TO_BYTE(F_B_OUT) + BOOL_TO_BYTE(F_C_OUT) + BOOL_TO_BYTE(F_D_OUT) + BOOL_TO_BYTE(F_E_OUT) + 1;
(* Network 13 *)
(* Network 14 *)
END_FUNCTION_BLOCK

(* POU BJ_FUWEI, LD *)
FUNCTION_BLOCK BJ_FUWEI
VAR_INPUT
	XH_A_SHUI: WORD;
	JQ_1: BOOL;
	JQ_2: BOOL;
	JQ_3: BOOL;
	JQ_4: BOOL;
	JQ_5: BOOL;
	JQ_6: BOOL;
END_VAR
VAR_OUTPUT
	FUWEI_A_OUT: BOOL;
	FS_KA: BOOL;
	JZ_OUT: BOOL;
END_VAR
VAR
	JT_A_SHU: WORD;

	FUWEI_A_3: BOOL;

	FUWEI_A_1: BOOL;

	FUWEI_A_2: BOOL;

	JQ_A_SHU: WORD;

END_VAR
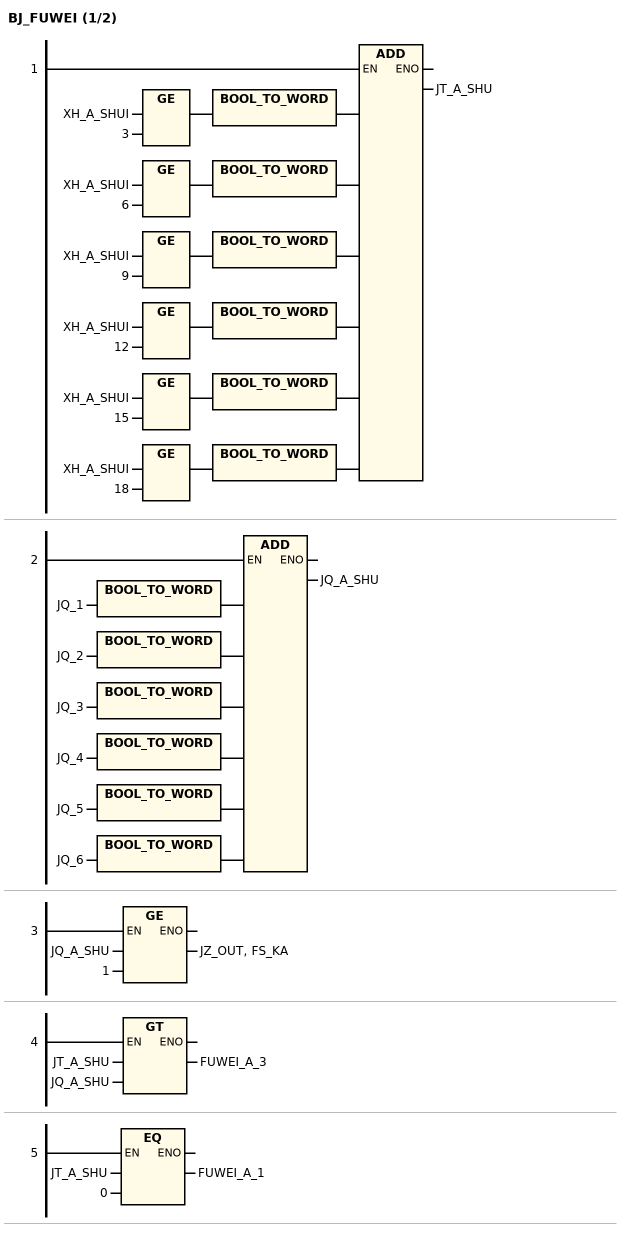
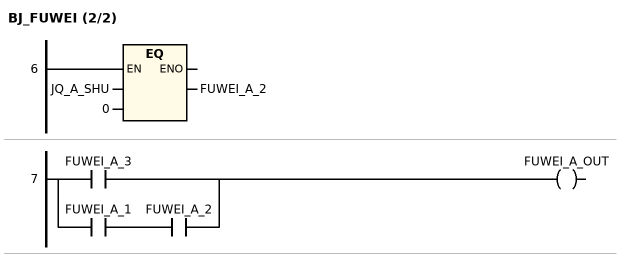
_LD_ (* Ladder Diagram *)
NETWORK 1
	*
		EN --- ADD(BOOL_TO_WORD(GE(XH_A_SHUI, 3)), BOOL_TO_WORD(GE(XH_A_SHUI, 6)), BOOL_TO_WORD(GE(XH_A_SHUI, 9)), BOOL_TO_WORD(GE(XH_A_SHUI, 12)), BOOL_TO_WORD(GE(XH_A_SHUI, 15)), BOOL_TO_WORD(GE(XH_A_SHUI, 18))) => JT_A_SHU
NETWORK 2
	*
		EN --- ADD(BOOL_TO_WORD(JQ_1), BOOL_TO_WORD(JQ_2), BOOL_TO_WORD(JQ_3), BOOL_TO_WORD(JQ_4), BOOL_TO_WORD(JQ_5), BOOL_TO_WORD(JQ_6)) => JQ_A_SHU
NETWORK 3
	*
		EN --- GE(JQ_A_SHU, 1) => JZ_OUT, FS_KA
NETWORK 4
	*
		EN --- GT(JT_A_SHU, JQ_A_SHU) => FUWEI_A_3
NETWORK 5
	*
		EN --- EQ(JT_A_SHU, 0) => FUWEI_A_1
NETWORK 6
	*
		EN --- EQ(JQ_A_SHU, 0) => FUWEI_A_2
NETWORK 7
	{ [FUWEI_A_3] | [FUWEI_A_1] - [FUWEI_A_2] } --- (FUWEI_A_OUT)
_END_LD_
(* the same logic as Structured Text *)
(* Network 1 *)
JT_A_SHU := BOOL_TO_WORD(XH_A_SHUI >= 3) + BOOL_TO_WORD(XH_A_SHUI >= 6) + BOOL_TO_WORD(XH_A_SHUI >= 9) + BOOL_TO_WORD(XH_A_SHUI >= 12) + BOOL_TO_WORD(XH_A_SHUI >= 15) + BOOL_TO_WORD(XH_A_SHUI >= 18);
(* Network 2 *)
JQ_A_SHU := BOOL_TO_WORD(JQ_1) + BOOL_TO_WORD(JQ_2) + BOOL_TO_WORD(JQ_3) + BOOL_TO_WORD(JQ_4) + BOOL_TO_WORD(JQ_5) + BOOL_TO_WORD(JQ_6);
(* Network 3: see the listing above *)
(* Network 4 *)
FUWEI_A_3 := JT_A_SHU > JQ_A_SHU;
(* Network 5 *)
FUWEI_A_1 := JT_A_SHU = 0;
(* Network 6 *)
FUWEI_A_2 := JQ_A_SHU = 0;
(* Network 7 *)
FUWEI_A_OUT := FUWEI_A_3 OR FUWEI_A_1 AND FUWEI_A_2;
END_FUNCTION_BLOCK

(* POU XH_PAIXU, LD *)
FUNCTION_BLOCK XH_PAIXU
VAR_INPUT
	XH_SHU_IN: WORD;
	ONE_CIXU: BYTE;
	TWO_CIXU: BYTE;
	THREE_CIXU: BYTE;
	FOUER_CIXU: BYTE;
	FIVE_CIXU: BYTE;
	SIX_CIXU: BYTE;
	XH_CLOSE_YSH: WORD;
	ON_OFF: BOOL;
END_VAR
VAR_OUTPUT
	ONE_OUT: BOOL;
	ONE_50_OUT: BOOL;
	ONE_75_OUT: BOOL;
	ONE_100_OUT: BOOL;
	TWO_OUT: BOOL;
 	TWO_50_OUT: BOOL;
	TWO_75_OUT: BOOL;
	TWO_100_OUT: BOOL;
	THREE_OUT: BOOL;
	THREE_50_OUT: BOOL;
	THREE_75_OUT: BOOL;
	THREE_100_OUT: BOOL;
	FOUER_OUT: BOOL;
	FOUER_50_OUT: BOOL;
	FOUER_75_OUT: BOOL;
	FOUER_100_OUT: BOOL;
	FIVE_OUT: BOOL;
	FIVE_50_OUT: BOOL;
	FIVE_75_OUT: BOOL;
	FIVE_100_OUT: BOOL;
	SIX_OUT: BOOL;
	SIX_50_OUT: BOOL;
	SIX_75_OUT: BOOL;
	SIX_100_OUT: BOOL;
END_VAR
VAR
	JQ_1: XH_PAIXU_1;
	JQ_2: XH_PAIXU_1;
	JQ_3: XH_PAIXU_1;
	JQ_4: XH_PAIXU_1;
	JQ_5: XH_PAIXU_1;
	JQ_6: XH_PAIXU_1;
END_VAR
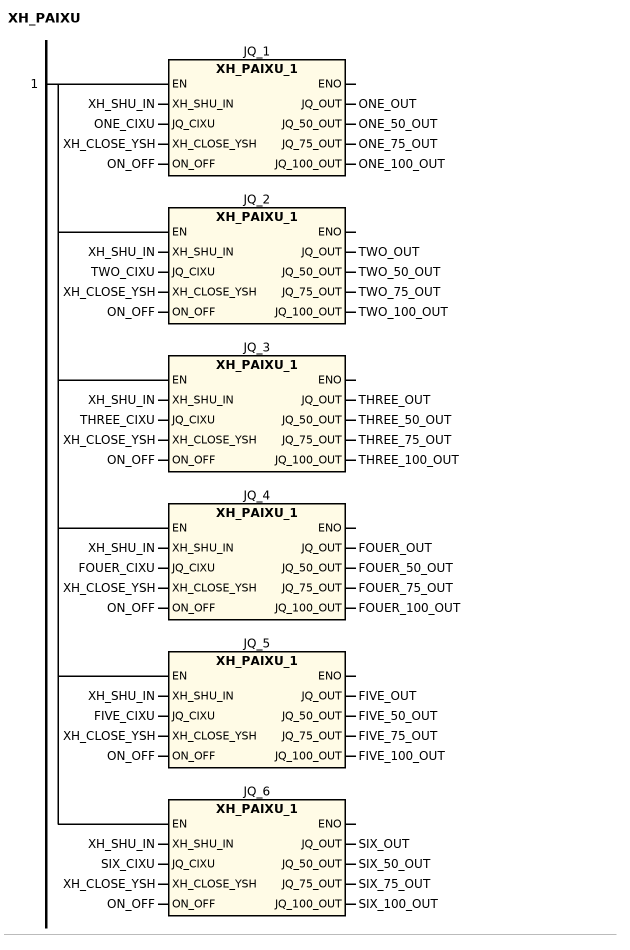
_LD_ (* Ladder Diagram *)
NETWORK 1
	*
		EN --- JQ_1:XH_PAIXU_1(XH_SHU_IN: XH_SHU_IN, JQ_CIXU: ONE_CIXU, XH_CLOSE_YSH: XH_CLOSE_YSH, ON_OFF: ON_OFF, JQ_50_OUT => ONE_50_OUT, JQ_75_OUT => ONE_75_OUT, JQ_100_OUT => ONE_100_OUT) => ONE_OUT
		EN --- JQ_2:XH_PAIXU_1(XH_SHU_IN: XH_SHU_IN, JQ_CIXU: TWO_CIXU, XH_CLOSE_YSH: XH_CLOSE_YSH, ON_OFF: ON_OFF, JQ_50_OUT => TWO_50_OUT, JQ_75_OUT => TWO_75_OUT, JQ_100_OUT => TWO_100_OUT) => TWO_OUT
		EN --- JQ_3:XH_PAIXU_1(XH_SHU_IN: XH_SHU_IN, JQ_CIXU: THREE_CIXU, XH_CLOSE_YSH: XH_CLOSE_YSH, ON_OFF: ON_OFF, JQ_50_OUT => THREE_50_OUT, JQ_75_OUT => THREE_75_OUT, JQ_100_OUT => THREE_100_OUT) => THREE_OUT
		EN --- JQ_4:XH_PAIXU_1(XH_SHU_IN: XH_SHU_IN, JQ_CIXU: FOUER_CIXU, XH_CLOSE_YSH: XH_CLOSE_YSH, ON_OFF: ON_OFF, JQ_50_OUT => FOUER_50_OUT, JQ_75_OUT => FOUER_75_OUT, JQ_100_OUT => FOUER_100_OUT) => FOUER_OUT
		EN --- JQ_5:XH_PAIXU_1(XH_SHU_IN: XH_SHU_IN, JQ_CIXU: FIVE_CIXU, XH_CLOSE_YSH: XH_CLOSE_YSH, ON_OFF: ON_OFF, JQ_50_OUT => FIVE_50_OUT, JQ_75_OUT => FIVE_75_OUT, JQ_100_OUT => FIVE_100_OUT) => FIVE_OUT
		EN --- JQ_6:XH_PAIXU_1(XH_SHU_IN: XH_SHU_IN, JQ_CIXU: SIX_CIXU, XH_CLOSE_YSH: XH_CLOSE_YSH, ON_OFF: ON_OFF, JQ_50_OUT => SIX_50_OUT, JQ_75_OUT => SIX_75_OUT, JQ_100_OUT => SIX_100_OUT) => SIX_OUT
_END_LD_
(* the same logic as Structured Text *)
(* Network 1 *)
JQ_1(XH_SHU_IN := XH_SHU_IN, JQ_CIXU := ONE_CIXU, XH_CLOSE_YSH := XH_CLOSE_YSH, ON_OFF := ON_OFF);
ONE_50_OUT := JQ_1.JQ_50_OUT;
ONE_75_OUT := JQ_1.JQ_75_OUT;
ONE_100_OUT := JQ_1.JQ_100_OUT;
ONE_OUT := JQ_1.JQ_OUT;
JQ_2(XH_SHU_IN := XH_SHU_IN, JQ_CIXU := TWO_CIXU, XH_CLOSE_YSH := XH_CLOSE_YSH, ON_OFF := ON_OFF);
TWO_50_OUT := JQ_2.JQ_50_OUT;
TWO_75_OUT := JQ_2.JQ_75_OUT;
TWO_100_OUT := JQ_2.JQ_100_OUT;
TWO_OUT := JQ_2.JQ_OUT;
JQ_3(XH_SHU_IN := XH_SHU_IN, JQ_CIXU := THREE_CIXU, XH_CLOSE_YSH := XH_CLOSE_YSH, ON_OFF := ON_OFF);
THREE_50_OUT := JQ_3.JQ_50_OUT;
THREE_75_OUT := JQ_3.JQ_75_OUT;
THREE_100_OUT := JQ_3.JQ_100_OUT;
THREE_OUT := JQ_3.JQ_OUT;
JQ_4(XH_SHU_IN := XH_SHU_IN, JQ_CIXU := FOUER_CIXU, XH_CLOSE_YSH := XH_CLOSE_YSH, ON_OFF := ON_OFF);
FOUER_50_OUT := JQ_4.JQ_50_OUT;
FOUER_75_OUT := JQ_4.JQ_75_OUT;
FOUER_100_OUT := JQ_4.JQ_100_OUT;
FOUER_OUT := JQ_4.JQ_OUT;
JQ_5(XH_SHU_IN := XH_SHU_IN, JQ_CIXU := FIVE_CIXU, XH_CLOSE_YSH := XH_CLOSE_YSH, ON_OFF := ON_OFF);
FIVE_50_OUT := JQ_5.JQ_50_OUT;
FIVE_75_OUT := JQ_5.JQ_75_OUT;
FIVE_100_OUT := JQ_5.JQ_100_OUT;
FIVE_OUT := JQ_5.JQ_OUT;
JQ_6(XH_SHU_IN := XH_SHU_IN, JQ_CIXU := SIX_CIXU, XH_CLOSE_YSH := XH_CLOSE_YSH, ON_OFF := ON_OFF);
SIX_50_OUT := JQ_6.JQ_50_OUT;
SIX_75_OUT := JQ_6.JQ_75_OUT;
SIX_100_OUT := JQ_6.JQ_100_OUT;
SIX_OUT := JQ_6.JQ_OUT;
END_FUNCTION_BLOCK

(* POU XH_PAIXU_1, LD *)
FUNCTION_BLOCK XH_PAIXU_1
VAR_INPUT
	XH_SHU_IN: WORD;
	JQ_CIXU: BYTE;
	XH_CLOSE_YSH: WORD;
	ON_OFF: BOOL;
END_VAR
VAR_OUTPUT
	JQ_OUT: BOOL;
	JQ_50_OUT: BOOL;
	JQ_75_OUT: BOOL;
	JQ_100_OUT: BOOL;
END_VAR
VAR
	XH_2: BOOL;










	ONE_1: BOOL;
	ONE_2: BOOL;
	ONE_3: BOOL;



	ONE_4: BOOL;

	CLOSE_ONE: YANSHI_CLOSE;

	ONE_OUT_4_KA: BOOL;

	ONE_OUT_3_KA: BOOL;
	ONE_OUT_2_KA: BOOL;








	ONE_OUT_1_KA: BOOL;
	JT_1_KA: BOOL;
	JT_2_KA: BOOL;
	JT_3_KA: BOOL;
	JT_4_KA: BOOL;
	XH_1: BOOL;
	XH_3: BOOL;
	XH_4: BOOL;
	XH_5: BOOL;
	XH_6: BOOL;
	XH_7: BOOL;
	XH_8: BOOL;
	XH_9: BOOL;
	XH_10: BOOL;
	XH_11: BOOL;
	XH_12: BOOL;
	XH_13: BOOL;
	XH_14: BOOL;
	XH_15: BOOL;

	JT_5_KA: BOOL;
	ONE_5: BOOL;
	ONE_OUT_5_KA: BOOL;
	XH_18: BOOL;
	JT_6_KA: BOOL;
	XH_16: BOOL;
	XH_17: BOOL;
	ONE_6: BOOL;
	ONE_OUT_6_KA: BOOL;
END_VAR
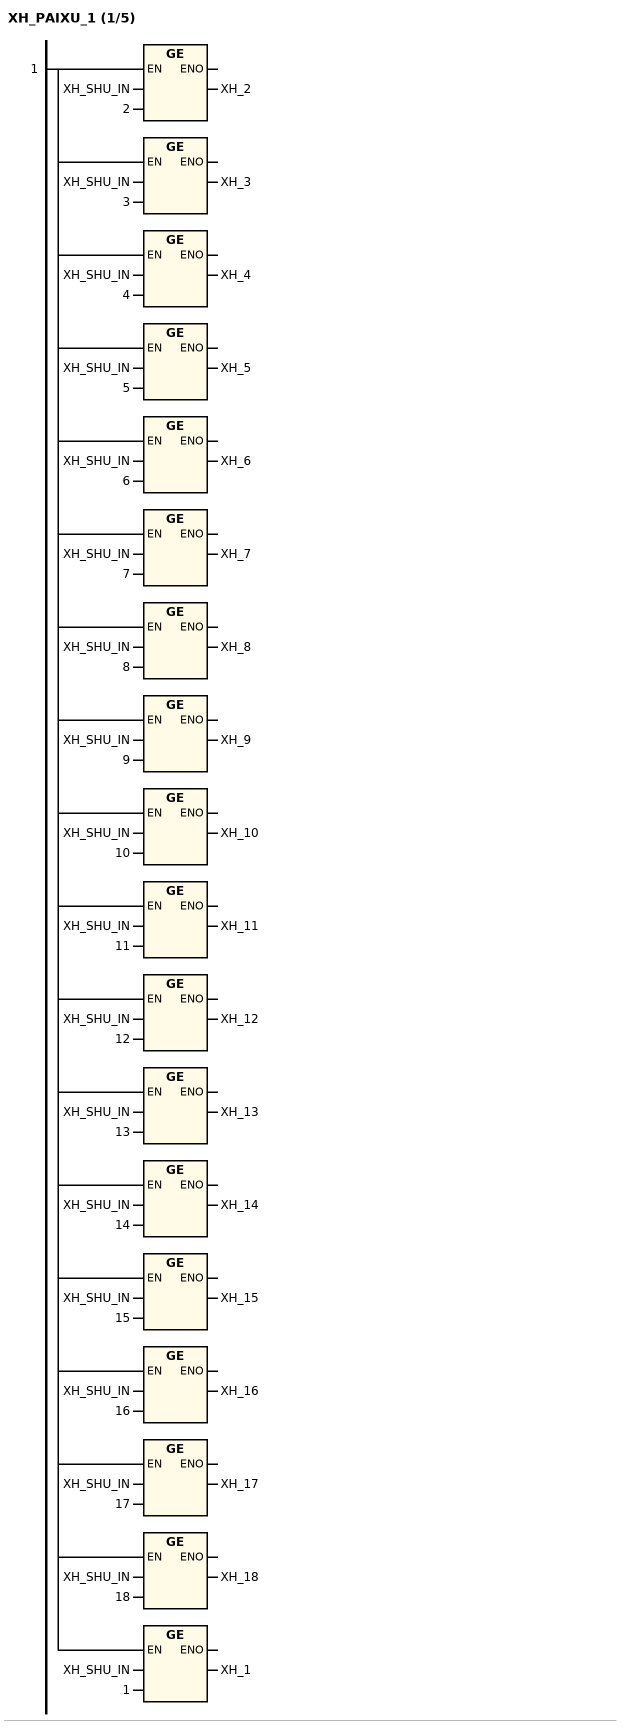
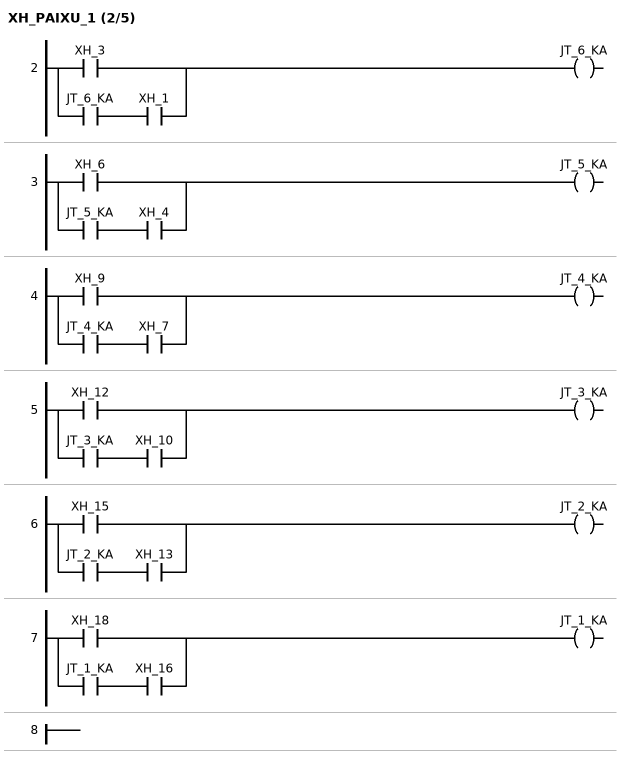
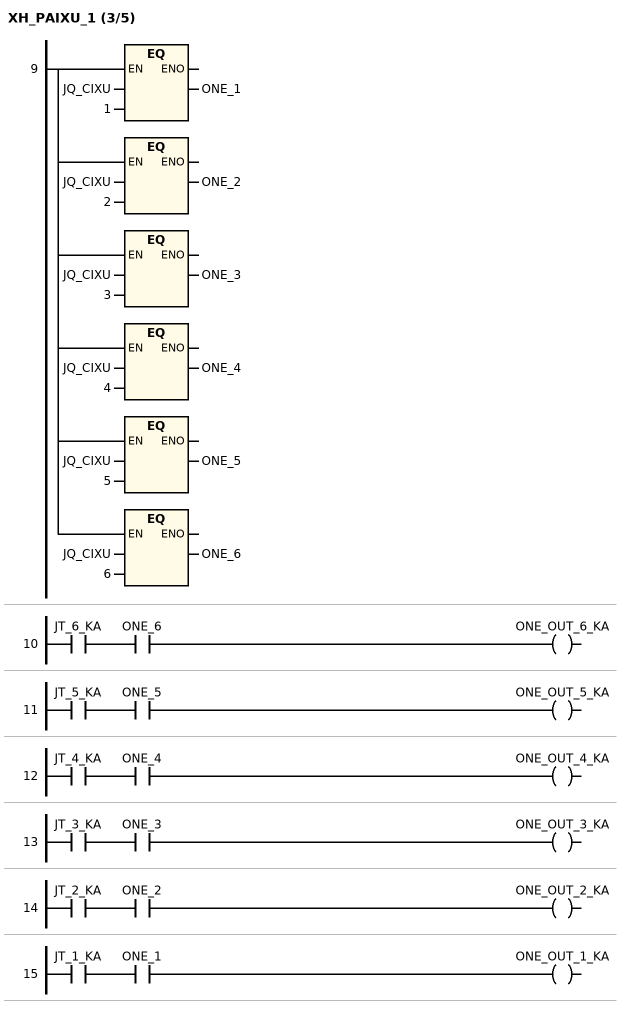
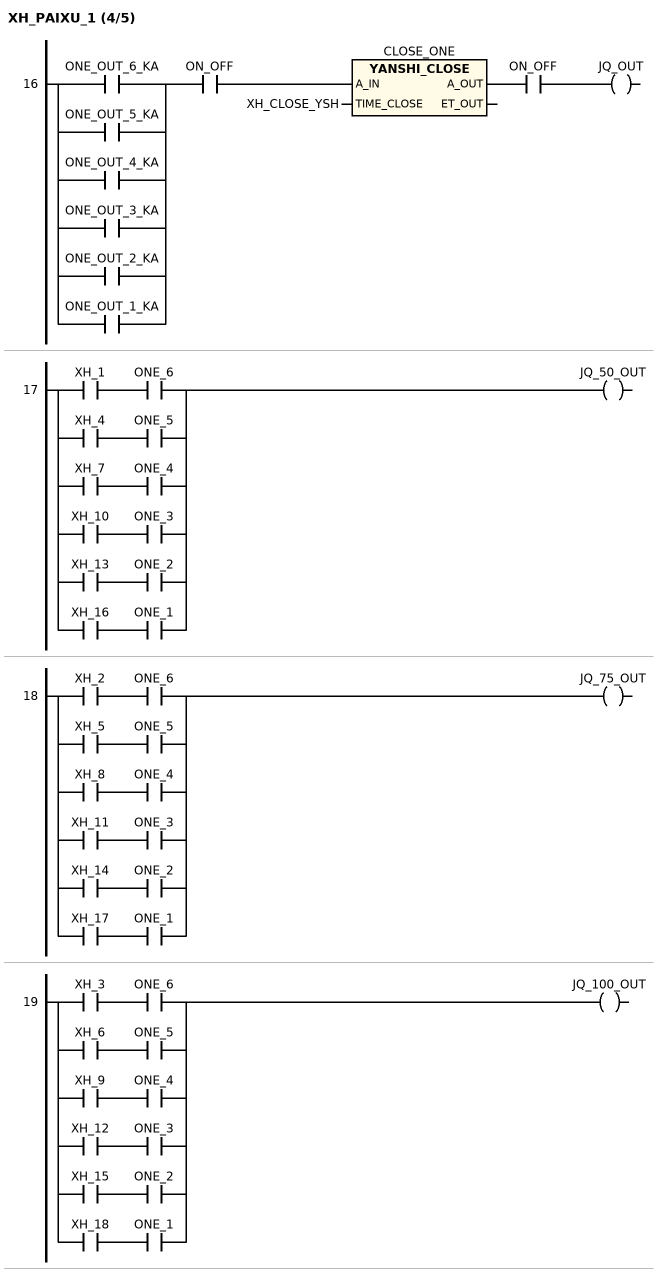
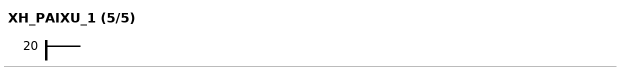
_LD_ (* Ladder Diagram *)
NETWORK 1
	*
		EN --- GE(XH_SHU_IN, 2) => XH_2
		EN --- GE(XH_SHU_IN, 3) => XH_3
		EN --- GE(XH_SHU_IN, 4) => XH_4
		EN --- GE(XH_SHU_IN, 5) => XH_5
		EN --- GE(XH_SHU_IN, 6) => XH_6
		EN --- GE(XH_SHU_IN, 7) => XH_7
		EN --- GE(XH_SHU_IN, 8) => XH_8
		EN --- GE(XH_SHU_IN, 9) => XH_9
		EN --- GE(XH_SHU_IN, 10) => XH_10
		EN --- GE(XH_SHU_IN, 11) => XH_11
		EN --- GE(XH_SHU_IN, 12) => XH_12
		EN --- GE(XH_SHU_IN, 13) => XH_13
		EN --- GE(XH_SHU_IN, 14) => XH_14
		EN --- GE(XH_SHU_IN, 15) => XH_15
		EN --- GE(XH_SHU_IN, 16) => XH_16
		EN --- GE(XH_SHU_IN, 17) => XH_17
		EN --- GE(XH_SHU_IN, 18) => XH_18
		EN --- GE(XH_SHU_IN, 1) => XH_1
NETWORK 2
	{ [XH_3] | [JT_6_KA] - [XH_1] } --- (JT_6_KA)
NETWORK 3
	{ [XH_6] | [JT_5_KA] - [XH_4] } --- (JT_5_KA)
NETWORK 4
	{ [XH_9] | [JT_4_KA] - [XH_7] } --- (JT_4_KA)
NETWORK 5
	{ [XH_12] | [JT_3_KA] - [XH_10] } --- (JT_3_KA)
NETWORK 6
	{ [XH_15] | [JT_2_KA] - [XH_13] } --- (JT_2_KA)
NETWORK 7
	{ [XH_18] | [JT_1_KA] - [XH_16] } --- (JT_1_KA)
NETWORK 8
	*
NETWORK 9
	*
		EN --- EQ(JQ_CIXU, 1) => ONE_1
		EN --- EQ(JQ_CIXU, 2) => ONE_2
		EN --- EQ(JQ_CIXU, 3) => ONE_3
		EN --- EQ(JQ_CIXU, 4) => ONE_4
		EN --- EQ(JQ_CIXU, 5) => ONE_5
		EN --- EQ(JQ_CIXU, 6) => ONE_6
NETWORK 10
	[JT_6_KA] - [ONE_6] --- (ONE_OUT_6_KA)
NETWORK 11
	[JT_5_KA] - [ONE_5] --- (ONE_OUT_5_KA)
NETWORK 12
	[JT_4_KA] - [ONE_4] --- (ONE_OUT_4_KA)
NETWORK 13
	[JT_3_KA] - [ONE_3] --- (ONE_OUT_3_KA)
NETWORK 14
	[JT_2_KA] - [ONE_2] --- (ONE_OUT_2_KA)
NETWORK 15
	[JT_1_KA] - [ONE_1] --- (ONE_OUT_1_KA)
NETWORK 16
	{ [ONE_OUT_6_KA] | [ONE_OUT_5_KA] | [ONE_OUT_4_KA] | [ONE_OUT_3_KA] | [ONE_OUT_2_KA] | [ONE_OUT_1_KA] } - [ON_OFF] - CLOSE_ONE:YANSHI_CLOSE(A_IN: *, TIME_CLOSE: XH_CLOSE_YSH) - [ON_OFF] --- (JQ_OUT)
NETWORK 17
	{ [XH_1] - [ONE_6] | [XH_4] - [ONE_5] | [XH_7] - [ONE_4] | [XH_10] - [ONE_3] | [XH_13] - [ONE_2] | [XH_16] - [ONE_1] } --- (JQ_50_OUT)
NETWORK 18
	{ [XH_2] - [ONE_6] | [XH_5] - [ONE_5] | [XH_8] - [ONE_4] | [XH_11] - [ONE_3] | [XH_14] - [ONE_2] | [XH_17] - [ONE_1] } --- (JQ_75_OUT)
NETWORK 19
	{ [XH_3] - [ONE_6] | [XH_6] - [ONE_5] | [XH_9] - [ONE_4] | [XH_12] - [ONE_3] | [XH_15] - [ONE_2] | [XH_18] - [ONE_1] } --- (JQ_100_OUT)
NETWORK 20
	*
_END_LD_
(* the same logic as Structured Text *)
(* Network 1 *)
XH_2 := XH_SHU_IN >= 2;
XH_3 := XH_SHU_IN >= 3;
XH_4 := XH_SHU_IN >= 4;
XH_5 := XH_SHU_IN >= 5;
XH_6 := XH_SHU_IN >= 6;
XH_7 := XH_SHU_IN >= 7;
XH_8 := XH_SHU_IN >= 8;
XH_9 := XH_SHU_IN >= 9;
XH_10 := XH_SHU_IN >= 10;
XH_11 := XH_SHU_IN >= 11;
XH_12 := XH_SHU_IN >= 12;
XH_13 := XH_SHU_IN >= 13;
XH_14 := XH_SHU_IN >= 14;
XH_15 := XH_SHU_IN >= 15;
XH_16 := XH_SHU_IN >= 16;
XH_17 := XH_SHU_IN >= 17;
XH_18 := XH_SHU_IN >= 18;
XH_1 := XH_SHU_IN >= 1;
(* Network 2 *)
JT_6_KA := XH_3 OR JT_6_KA AND XH_1;
(* Network 3 *)
JT_5_KA := XH_6 OR JT_5_KA AND XH_4;
(* Network 4 *)
JT_4_KA := XH_9 OR JT_4_KA AND XH_7;
(* Network 5 *)
JT_3_KA := XH_12 OR JT_3_KA AND XH_10;
(* Network 6 *)
JT_2_KA := XH_15 OR JT_2_KA AND XH_13;
(* Network 7 *)
JT_1_KA := XH_18 OR JT_1_KA AND XH_16;
(* Network 8 *)
(* Network 9 *)
ONE_1 := JQ_CIXU = 1;
ONE_2 := JQ_CIXU = 2;
ONE_3 := JQ_CIXU = 3;
ONE_4 := JQ_CIXU = 4;
ONE_5 := JQ_CIXU = 5;
ONE_6 := JQ_CIXU = 6;
(* Network 10 *)
ONE_OUT_6_KA := JT_6_KA AND ONE_6;
(* Network 11 *)
ONE_OUT_5_KA := JT_5_KA AND ONE_5;
(* Network 12 *)
ONE_OUT_4_KA := JT_4_KA AND ONE_4;
(* Network 13 *)
ONE_OUT_3_KA := JT_3_KA AND ONE_3;
(* Network 14 *)
ONE_OUT_2_KA := JT_2_KA AND ONE_2;
(* Network 15 *)
ONE_OUT_1_KA := JT_1_KA AND ONE_1;
(* Network 16 *)
CLOSE_ONE(A_IN := (ONE_OUT_6_KA OR ONE_OUT_5_KA OR ONE_OUT_4_KA OR ONE_OUT_3_KA OR ONE_OUT_2_KA OR ONE_OUT_1_KA) AND ON_OFF, TIME_CLOSE := XH_CLOSE_YSH);
JQ_OUT := CLOSE_ONE.A_OUT AND ON_OFF;
(* Network 17 *)
JQ_50_OUT := XH_1 AND ONE_6 OR XH_4 AND ONE_5 OR XH_7 AND ONE_4 OR XH_10 AND ONE_3 OR XH_13 AND ONE_2 OR XH_16 AND ONE_1;
(* Network 18 *)
JQ_75_OUT := XH_2 AND ONE_6 OR XH_5 AND ONE_5 OR XH_8 AND ONE_4 OR XH_11 AND ONE_3 OR XH_14 AND ONE_2 OR XH_17 AND ONE_1;
(* Network 19 *)
JQ_100_OUT := XH_3 AND ONE_6 OR XH_6 AND ONE_5 OR XH_9 AND ONE_4 OR XH_12 AND ONE_3 OR XH_15 AND ONE_2 OR XH_18 AND ONE_1;
(* Network 20 *)
END_FUNCTION_BLOCK

(* POU DY_JT_KZH, LD *)
FUNCTION_BLOCK DY_JT_KZH
VAR_INPUT
	TD_TON_IN: BOOL;
	DY_BH_IN: BOOL;
	JT_IN: BOOL;
	REST: BOOL;
END_VAR
VAR_OUTPUT
	DY_BH_OUT: BOOL;
	JT_OUT: BOOL;
	DY_BH_ET: WORD;
	HM_OUT: WORD;
	DY_JT_OUT: BOOL;
END_VAR
VAR
	DY_FW: BOOL;
	DY_OPEN: YANSHI_OPEN;

	DY_R: R_TRIG;
	JT_R: R_TRIG;
	KJ_TON: TON;
	DY_TON: TON;
	JT_TON: TON;
	KJ_SUO: BOOL;
	DY_SUO: BOOL;
	JT_SUO: BOOL;
	KJ_R: R_TRIG;
END_VAR
VAR_IN_OUT
	DY_FW_SET: WORD;
END_VAR
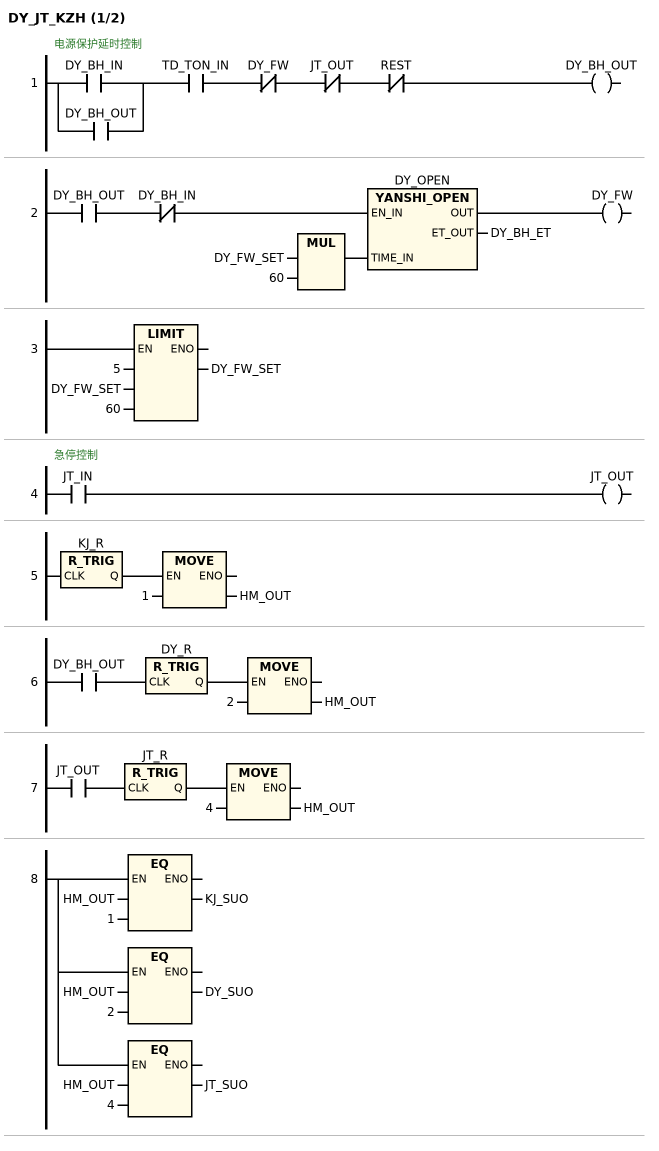
